Universal Robots PolyScope program: AutoGrind02.urp

Program AutoGrind02 (installation=default directory=/programs/AutoGrind createdIn=5.7.0.90932 lastSavedIn=5.11.11.1010533 robotSerialNumber=20195501059)
Calibrated DH parameters: a=[0.000146, -0.418764, -0.053981, 0.000058, -0.000023, 0]; d=[0.162545, 37.319448, -206.067439, 168.881546, 0.09955, 0.099464]; alpha=[1.57004, -0.001979, 0.002304, 1.570607, -1.57066, 0]; deltaTheta=[0, -0.174616, -1.258233, 1.432844, -0.000001, 0]
BeforeStart
  Script file /programs/AutoGrind/agscript_util-2.script
    | # File: agscript_util-2.scripts
    | # Project: AutoGrind
    | # Author: Ned Lecky, Lecky Engineering LLC
    | # Purpose: General utility function used in AutoGrind
    | 
    | global robot_util_version = "Rev 2 2022-06-02"
    | 
    | # Return max of 2 numeric values
    | def max(n1, n2):
    |   if n1 > n2:
    |     return n1
    |   else:
    |     return n2
    |   end
    | end
    | 
    | # Return min of 2 numeric values
    | def min(n1, n2):
    |   if n1 < n2:
    |     return n1
    |   else:
    |     return n2
    |   end
    | end
    | 
    | # Return absolute value of a numeric value
    | def abs(n):
    |   if n < 0:
    |     return -n
    |   else:
    |     return n
    |   end
    | end
    | 
    | # Return param limited to lowLim <= param <= hiLim
    | def limiter(param, loLim, hiLim):
    |   if param < loLim:
    |     return loLim
    |   elif param > hiLim:
    |     return hiLim
    |   else:
    |     return param
    |   end
    | end
    | 
    | # Send LF out the socket
    | def socket_send_lf():
    |   socket_send_byte(10)
    | end
    | 
    | # Send n-vectors back to socket as [n,n,n,n,n,n]
    | def return_vector(p, n = 6):
    |   socket_send_string("[")
    |   i = 0
    |   while i < n:
    |     if i > 0:
    |       socket_send_string(",")
    |     end
    |     socket_send_string(p[i])
    |     i = i + 1
    |   end
    |   socket_send_string("]")
    | end
    | 
    | # Send 6-element position back to socket as:
    | #   (isPose=False)  name=[n,n,n,n,n,n]
    | #   (isPose=True)   name=p[n,n,n,n,n,n]
    | def return_position(name, isPose, p):
    |   socket_send_string(name)
    |   socket_send_string("=")
    |   if isPose == True:
    |     socket_send_string("p")
    |   end
    |   return_vector(p, 6)
    |   socket_send_lf()
    | end
    | 
    | # Return a 6-element vector to socket as a pose name=p[.....]
    | def return_pose(name, p):
    |   return_position(name, True, p)
    | end
    | 
    | # Return a 6-element vector to socket as joint angles name=[.....]
    | def return_joints(name, p):
    |   return_position(name, False, p)
    | end
    | 
    | # Special support to receive 1-4 port,value pairs and always pad with -1s to make 4 pairs
    | # Essentialy returns command[3:end] padded out with -1s to always be 8 elements
    | # Assumes length of command is specified in command[0]
    | def command_3_padded_8(command):
    |   ret8 = [-1, -1, -1, -1, -1, -1, -1, -1]
    |   i = 0
    |   while i < command[0]-2:
    |     ret8[i] = command[i + 3]
    |     i = i + 1
    |   end
    |   return ret8
    | end
  Script file /programs/AutoGrind/agscript_robot-2.script
    | # File: agscript_robot-2.script
    | # Project: AutoGrind
    | # Author: Ned Lecky, Lecky Engineering LLC
    | # Purpose: Robot control commands supporting the AutoGrind application
    | 
    | global robot_version = "Rev 2 2022-06-07"
    | 
    | global response = "unknown"
    | global robot_index = 0
    | global robot_checkvalue = 0
    | 
    | global robot_linear_speed_mps = 0.2
    | global robot_linear_accel_mpss = 0.4
    | global robot_blend_radius_m = 0.003
    | global robot_joint_speed_rps = 1.0
    | global robot_joint_accel_rpss = 4.0
    | global robot_tcp = p[0, 0, 0.175, 0, 0, 0]
    | global robot_tcp_part = robot_tcp
    | global robot_payload_mass_kg = 1.0
    | global robot_payload_cog_m = [0, 0, 0.50]
    | # Geometry [1=FLAT 2=CYL 3=SPHERE, diameter_mm)
    | global robot_part_geometry = [0, 0]
    | global robot_door_closed_input = [-1, -1]
    | global robot_footswitch_pressed_input = [-1, -1]
    | global robot_tool_on_outputs = [-1, -1, -1, -1, -1, -1, -1, -1]
    | global robot_tool_off_outputs = [-1, -1, -1, -1, -1, -1, -1, -1]
    | global robot_coolant_on_outputs = [-1, -1, -1, -1, -1, -1, -1, -1]
    | global robot_coolant_off_outputs = [-1, -1, -1, -1, -1, -1, -1, -1]
    | global robot_freedrive_mode = 0
    | 
    | # command should be[nElements,index,checkval,param[0],param[1],...]
    | # put index into robot_index
    | # validate checkval
    | # Remove both from command so we get command = [nElements-2, param[0], param[1],...]
    | #global command = [0., 0., 0., 0., 0., 0., 0., 0., 0., 0., 0., 0., 0.]
    | def command_validate():
    |   # must be at least index, check, and 1 param
    |   if command[0] < 3:
    |     command[0] = 0
    |     return False
    |   end
    | 
    |   # Now make sure checksum matches what we expect
    |   global test_index = command[1]
    |   global test_checksum = command[2]
    |   if test_checksum != 1000 - test_index:
    |     command[0] = 0
    |     return False
    |   end
    | 
    |   # Now if we are still in the grind state and we are not getting a grind command (40) make sure we're are off the part!
    |   if grind_process_state and command[3] != 40:
    |     # Using set_grind_process_state which assumes robot_tcp_part!
    |     iset_tcp(robot_tcp_part)
    |     set_grind_process_state(False)
    |     iset_tcp(robot_tcp)
    |   end
    | 
    |   # Slide the robot commands and parameters back in command[] to remove the index and checksum
    |   local i = 3
    |   while (i < command[0] + 1):
    |     command[i-2] = command[i]
    |     i = i + 1
    |   end
    |   command[i-1] = 0
    |   command[i-2] = 0
    |   command[0] = command[0] - 2    # 2 fewer elements in the array now!
    | 
    |   global robot_index = test_index
    |   return True
    | end
    | 
    | # Call this when starting command execution
    | def command_start():
    |   global last_comand = command
    | 
    |   # This one signifies we're starting a new command!
    |   global robot_starting = robot_index
    |   socket_set_var("robot_starting", robot_starting)
    |   socket_send_line("robot_ready=False")
    | end
    | 
    | # Call this when a command is complete
    | def command_finish():
    |   local retval = "robot_response=" + response + "#robot_ready=True"
    |   socket_send_line(retval)
    | 
    |   global robot_completed = robot_index
    |   socket_set_var("robot_completed", robot_completed)
    | end
    | 
    | # Set variable interface. Interprets command[2] to select what to set and returns result to socket
    | # Can also be used for validation and enforcing limits
    | def set_variable():
    |   if command[2] == 1:
    |     # Set speed to s if s>0. Always returns current value
    |     s = command[3]
    |     if s > 0:
    |       robot_linear_speed_mps = ceil(s) / 1000.0
    |     end
    |     socket_set_var("robot_linear_speed_mmps", robot_linear_speed_mps * 1000.0)
    |     global response = "set_linear_speed()"
    |   elif command[2] == 2:
    |     # Set accel to a if a>0. Always returns current value
    |     a = command[3]
    |     if a > 0:
    |       robot_linear_accel_mpss = ceil(a) / 1000.0
    |     end
    |     socket_set_var("robot_linear_accel_mmpss", robot_linear_accel_mpss * 1000.0)
    |     global response = "set_linear_accel()"
    |   elif command[2] == 3:
    |     # Set blend to b if b>=0. Always returns current value
    |     b = command[3]
    |     if b >= 0:
    |       robot_blend_radius_m = b / 1000.0
    |     end
    |     socket_send_string("robot_blend_radius_mm=")
    |     socket_send_string(robot_blend_radius_m * 1000.0)
    |     socket_send_lf()
    |     global response = "set_blend_radius()"
    |   elif command[2] == 4:
    |     # Set joint speed to s if s>0. Always returns current value
    |     s = command[3]
    |     if s > 0:
    |       robot_joint_speed_rps = d2r(ceil(s))
    |     end
    |     socket_set_var("robot_joint_speed_dps", r2d(robot_joint_speed_rps))
    |     global response = "set_joint_speed()"
    |   elif command[2] == 5:
    |     # Set joint accel to a if a>0. Always returns current value
    |     a = command[3]
    |     if a > 0:
    |       robot_joint_accel_rpss = d2r(ceil(a))
    |     end
    |     socket_set_var("robot_joint_accel_dpss", r2d(robot_joint_accel_rpss))
    |     global response = "set_joint_accel()"
    |   elif command[2] == 6:
    |     # Set part_geometry to [shape, diameter_mm] if shape==1,2,3. Always returns "robot_part_geometry=[current geometry]"
    |     # Also updates robot_part_tcp using update_robot_tcp_part
    |     shape = command[3]
    |     if shape == 1:
    |       robot_part_geometry = [1, 0]
    |     elif shape == 2 or shape == 3:
    |       diameter_mm = limiter(command[4], 50, 3000)
    |       robot_part_geometry = [shape, diameter_mm]
    |     end
    | 
    |     update_robot_tcp_part()
    | 
    |     socket_send_string("robot_part_geometry=")
    |     return_vector(robot_part_geometry, 2)
    |     socket_send_lf()
    |     global response = "set_part_geometry()"
    |   elif command[2] == 10:
    |     # Set door closed input
    |     if command[3] >= 0:
    |       robot_door_closed_input[0] = command[3]
    |       robot_door_closed_input[1] = command[4]
    |     end
    | 
    |     socket_send_string("robot_door_closed_input=")
    |     return_vector(robot_door_closed_input, 2)
    |     socket_send_lf()
    |     socket_set_var("robot_door_closed", is_door_closed())
    |     global response = "set_door_closed_input()"
    |   elif command[2] == 11:
    |     # Set tool on output
    |     robot_tool_on_outputs = command_3_padded_8(command)
    | 
    |     socket_send_string("robot_tool_on_outputs=")
    |     return_vector(robot_tool_on_outputs, 8)
    |     socket_send_lf()
    |     global response = "set_tool_on_outputs()"
    |   elif command[2] == 12:
    |     # Set tool off output
    |     robot_tool_off_outputs = command_3_padded_8(command)
    | 
    |     socket_send_string("robot_tool_off_outputs=")
    |     return_vector(robot_tool_off_outputs, 8)
    |     socket_send_lf()
    |     global response = "set_tool_off_outputs()"
    |   elif command[2] == 13:
    |     # Set coolant on output
    |     robot_coolant_on_outputs = command_3_padded_8(command)
    | 
    |     socket_send_string("robot_coolant_on_outputs=")
    |     return_vector(robot_coolant_on_outputs, 8)
    |     socket_send_lf()
    |     global response = "set_coolant_on_outputs()"
    |   elif command[2] == 14:
    |     # Set coolant off output
    |     robot_coolant_off_outputs = command_3_padded_8(command)
    | 
    |     socket_send_string("robot_coolant_off_outputs=")
    |     return_vector(robot_coolant_off_outputs, 8)
    |     socket_send_lf()
    |     global response = "set_coolant_off_outputs()"
    |   elif command[2] == 15:
    |     # tool_on
    |     tool_power(True, 2)
    |     global response = "tool_on()"
    |   elif command[2] == 16:
    |     # tool_off
    |     tool_power(False, 2)
    |     global response = "tool_off()"
    |   elif command[2] == 17:
    |     # coolant_on
    |     coolant_flow(True, 2)
    |     global response = "coolant_on()"
    |   elif command[2] == 18:
    |     # coolant_off
    |     coolant_flow(False, 2)
    |     global response = "coolant_off()"
    |   elif command[2] == 19:
    |     # freedrive 1=on/0=off, 0=base|1=tcp|2=tcp_part, 6 axisEnables
    |     if command[3] == 0:
    |       end_freedrive_mode()
    |       iset_tcp(robot_tcp)
    |       robot_freedrive_mode = 0
    |       socket_set_var("robot_freedrive_mode", robot_freedrive_mode)
    |     else:
    |       local coordSys = command[4]
    |       local freeAxes = [command[5], command[6], command[7], command[8], command[9], command[10]]
    |       if coordSys == 1:
    |         iset_tcp(robot_tcp)
    |         freedrive_mode(freeAxes = freeAxes, feature = "tool")
    |       elif coordSys == 2:
    |         iset_tcp(robot_tcp_part)
    |         freedrive_mode(freeAxes = freeAxes, feature = "tool")
    |       else:
    |         # Base
    |         freedrive_mode(freeAxes = freeAxes)
    |       end
    |       robot_freedrive_mode = 1
    |       socket_set_var("robot_freedrive_mode", robot_freedrive_mode)
    |     end
    |     global response = "freedrive_mode()"
    |   elif command[2] == 20:
    |     # set_tcp if command[3] > -10. Always returns robot_tcp=p[...]
    |     if command[3] > -10:
    |       robot_tcp = p[command[3], command[4], command[5], command[6], command[7], command[8]]
    |       iset_tcp(robot_tcp)
    |     end
    |     return_pose("robot_tcp", get_tcp_offset())
    |     # Recompute robot_tcp_part based on current geometry
    |     update_robot_tcp_part()
    |     global response = "set_tcp()"
    |   elif command[2] == 21:
    |     # set_payload if command[3] > 0. Always return robot_m and robot_cog
    |     if command[3] > 0:
    |       robot_payload_mass_kg = command[3]
    |       robot_payload_cog_m = [command[4], command[5], command[6]]
    |       iset_payload(robot_payload_mass_kg, robot_payload_cog_m)
    |     end
    |     socket_set_var("robot_payload_mass_kg", robot_payload_mass_kg)
    |     socket_send_string("robot_payload_cog_m=")
    |     return_vector(robot_payload_cog_m, 3)
    |     socket_send_lf()
    |     global response = "set_payload()"
    |   elif command[2] == 22:
    |     # Set footswitch pressed input
    |     if command[3] >= 0:
    |       robot_footswitch_pressed_input[0] = command[3]
    |       robot_footswitch_pressed_input[1] = command[4]
    |     end
    | 
    |     socket_send_string("robot_footswitch_pressed_input=")
    |     return_vector(robot_footswitch_pressed_input, 2)
    |     socket_send_lf()
    |     socket_set_var("robot_footswitch_pressed", is_footswitch_pressed())
    |     global response = "set footswitch_pressed_input()"
    |   elif command[2] == 30:
    |     # set_output
    |     local out = command[3]
    |     local state = command[4] > 0
    |     set_digital_out(out, state)
    |     global response = "set_output()"
    |   else:
    |     global response = "set_variable ERROR"
    |   end
    | end
    | 
    | # Compute appropriate robot_tcp for the part based on robot_tcp and robot_part_geometry
    | # They're the same for flat parts, but the TCP is adjusted to the center of the cylinder or sphere
    | def update_robot_tcp_part():
    |   shape = robot_part_geometry[0]
    |   if shape == 1:  # Flat
    |     robot_tcp_part = robot_tcp
    |   else:  # Cylinder or Sphere
    |     robot_tcp_part = pose_trans(robot_tcp, p[0, 0, robot_part_geometry[1] / 2000.0, 0, 0, 0])
    |   end
    |   return_pose("robot_tcp_part", robot_tcp_part)
    | end
    | 
    | # Send get_tcp_offset() result to socket
    | def return_tcp_offset():
    |   p = get_tcp_offset()
    |   return_pose("tcp_offset", p)
    |   global response = "return_tcp_offset()"
    | end
    | 
    | # Send get_actual_tcp_pose() to socket
    | def return_actual_tcp_pose():
    |   p = iget_actual_tcp_pose()
    |   return_pose("actual_tcp_pose", p)
    |   global response = "return_actual_tcp_pose()"
    | end
    | 
    | # Send get_actual_joint_positions() to socket
    | def return_get_actual_joint_positions():
    |   p = iget_actual_joint_positions()
    |   return_joints("actual_joint_positions", p)
    |   global response = "return_get_actual_joint_positions()"
    | end
    | 
    | # Send both joints and pose to socket labeled position_p and position_q
    | def return_both_positions():
    |   return_joints("position_q", iget_actual_joint_positions())
    |   return_pose("position_p", iget_actual_tcp_pose())
    |   global response = "return_both_positions()"
    | end
    | 
    | # Movel relatively in base coordinates
    | def movel_relative_base(p1):
    |   local p0 = get_target_tcp_pose()
    |   local p2 = pose_add(p0, p1)
    |   if p1[0] == 0 and p1[1] == 0 and p1[2] == 0:  # Rotational move
    |     imovel(p2, robot_joint_accel_rpss, robot_joint_speed_rps)
    |   else:
    |     imovel(p2, robot_linear_accel_mpss, robot_linear_speed_mps)
    |   end
    |   global response = "movel_relative_base()"
    | end
    | 
    | # Movel relatively in TCP coordinates
    | def movel_relative_tcp(p1):
    |   local p2 = pose_trans(get_target_tcp_pose(), p1)
    |   if p1[0] == 0 and p1[1] == 0 and p1[2] == 0:  # Rotational move
    |     imovel(p2, robot_joint_accel_rpss, robot_joint_speed_rps)
    |   else:
    |     imovel(p2, robot_linear_accel_mpss, robot_linear_speed_mps)
    |   end
    |   global response = "movel_relative_tcp()"
    | end
    | 
    | # Movel relatively in TCP_part coordinates
    | def movel_relative_tcp_part(p1):
    |   iset_tcp(robot_tcp_part)
    |   local p2 = pose_trans(get_target_tcp_pose(), p1)
    |   if p1[0] == 0 and p1[1] == 0 and p1[2] == 0:  # Rotational move
    |     imovel(p2, robot_joint_accel_rpss, robot_joint_speed_rps)
    |   else:
    |     imovel(p2, robot_linear_accel_mpss, robot_linear_speed_mps)
    |   end
    |   iset_tcp(robot_tcp)
    |   global response = "movel_relative_tcp_part()"
    | end
    | 
    | # Change one element of current pose and movel there
    | def movel_one_only(index = 0, val = 0):
    |   local p = get_target_tcp_pose()
    |   p[index] = val
    |   if index < 3:  # Translational
    |     imovel(p, a = robot_linear_accel_mpss, v = robot_linear_speed_mps)
    |   else:
    |     imovel(p, a = robot_joint_accel_rpss, v = robot_joint_speed_rps)
    |   end
    |   global response = "movel_one_only()"
    | end
    | 
    | # Change only rotation elements of current pose and movel there
    | def movel_rot_only(r1 = 0, r2 = 0, r3 = 0):
    |   local p = get_target_tcp_pose()
    |   p[3] = r1
    |   p[4] = r2
    |   p[5] = r3
    |   imovel(p, a = robot_joint_accel_rpss, v = robot_joint_speed_rps)
    |   global response = "movel_rot_only()"
    | end
    | 
    | # Movej to position (works with joints or poses)
    | def movej_ag(p):
    |   imovej(p, a = robot_joint_accel_rpss, v = robot_joint_speed_rps)
    |   global response = "movej_ag()"
    | end
    | 
    | # Movel to position (works with joints or poses)
    | def movel_ag(p):
    |   imovel(p, a = robot_linear_accel_mpss, v = robot_linear_speed_mps)
    |   global response = "movel_ag()"
    | end
    | 
    | # ####################################################################################
    | # Interrupting Motion
    | # Motion and force_mode and part contact muct all end if any of 3 things happen
    | #  1) Door is opened
    | #  2) We're in contact with the part and grinding, but no grind command comes within some time (default 1.5s)
    | #  3) We receive an abort message from the host
    | #
    | # How is it implemented?
    | #
    | # 1) io_monitor_thread (below) is ALWAYS running. Fires every time_door_check_rate_s (0.25s)
    | #    - Whenever it sees the state of the door change, it sends SET robot_door_closed state to host
    | #    - Whenever it sees the state of the footswitch (DIN7) change, it sends SET robot_footswitch state to host
    | #    - It monitors if we're still in contact wth the part butr not grinding (grind_process_state and grind_ready)
    | #      - If that goes beyond grind_max_wait_ms it sets halt_grind=True
    | # 2) no_command function (below). Called by PolScript everyu time it's waiting for a command and doesn't get one with a second
    | #    - If halt_grind is set (by door monitor thread above)
    | #      - stopl and simulate receiving a grind_retract
    | #      - THIS FORCES THE force_off and motion commands to come from the primary thread, as they must
    | # 3) listener_thread started by grind()
    | #    - This runs only while a grind is in progress
    | #    - It listens for commands from the host since PolyScope is blocked
    | #    - Any command received increments halt_count which makes ok_to_proceed() false
    | #    - That is checked in all the grinding programs and forces them to finish up and get off the part in an orderly fashion
    | 
    | # ####################################################################################
    | # START AUTOMATED DOOR MONITORING THREAD
    | #
    | # Return True if door in closed state (or if door input is undefined)
    | def is_door_closed():
    |   if robot_door_closed_input[0] < 0:
    |     return True
    |   end
    |   if get_standard_digital_in(robot_door_closed_input[0]):
    |     f = 1
    |   else:
    |     f = 0
    |   end
    |   return f == robot_door_closed_input[1]
    | end
    | 
    | # Return True if footswitch pressed (or False if footswitch input is undefined)
    | def is_footswitch_pressed():
    |   if robot_footswitch_pressed_input[0] < 0:
    |     return False
    |   end
    |   if get_standard_digital_in(robot_footswitch_pressed_input[0]):
    |     f = 1
    |   else:
    |     f = 0
    |   end
    |   return f == robot_footswitch_pressed_input[1]
    | end
    | 
    | global robot_door_closed = is_door_closed()
    | global robot_footswitch_pressed = is_footswitch_pressed()
    | global time_in_uncommanded_grind = 0
    | global time_door_check_rate_s = 0.250
    | global grind_max_wait_ms = 1500
    | # Also monitors footswitch!
    | thread io_monitor_thread():
    |   # Send current state on start... in future will only be sent on change
    |   socket_set_var("robot_door_closed", robot_door_closed)
    |   socket_set_var("robot_footswitch_pressed", robot_footswitch_pressed)
    | 
    |   while True:
    |     sleep(time_door_check_rate_s)
    |     local new_door_closed = is_door_closed()
    |     local new_footswitch_pressed = is_footswitch_pressed()
    | 
    |     # Notify host if door state has changed
    |     if robot_door_closed != new_door_closed:
    |       robot_door_closed = new_door_closed
    |       socket_set_var("robot_door_closed", robot_door_closed)
    |     end
    | 
    |     # Notify host if footswitch state has changed
    |     if robot_footswitch_pressed != new_footswitch_pressed:
    |       robot_footswitch_pressed = new_footswitch_pressed
    |       socket_set_var("robot_footswitch_pressed", robot_footswitch_pressed)
    |     end
    | 
    |     # Check for still in grind process but not executing a grind command
    |     # This is what happens after a grind_...(....,1) executes while waiting for next command
    |     if grind_process_state and grind_ready:
    |       time_in_uncommanded_grind = time_in_uncommanded_grind + time_door_check_rate_s
    |       # No new grind commands for grind_max_wait_ms... schedule a grind_retract!
    |       if time_in_uncommanded_grind > grind_max_wait_ms / 1000.0:
    |         global halt_grind = True
    |       end
    |     else:
    |       time_in_uncommanded_grind = 0
    |     end
    |   end
    | end
    | global ioMonitorThread = run io_monitor_thread()
    | #
    | # END AUTOMATED DOOR MONITORING THREAD
    | # ####################################################################################
    | 
    | # ####################################################################################
    | # START NO_COMMAND HOUSEKEEPING
    | # This gets called when the PolyScope receives no command (about 1/second)
    | # We can fire off any command here safely since no others will be seen until we exit
    | #
    | global no_command_count = 0
    | global halt_grind = False
    | def no_command():
    |   global no_command_count = no_command_count + 1
    | 
    |   if grind_process_state and grind_ready and halt_grind:
    |     halt_grind = False
    |     istopl(20)
    | 
    |     iset_tcp(robot_tcp_part)
    |     set_grind_process_state(False)
    |     iset_tcp(robot_tcp)
    |   end
    | end
    | #
    | # END NO_COMMAND HOUSEKEEPING
    | # ####################################################################################
    | 
    | # ####################################################################################
    | # START TOUCHOFF HANDLER
    | #
    | def calculate_point_to_move_towards(feature, direction, position_distance):
    |   local posDir = [direction[0], direction[1], direction[2]]
    |   if (norm(posDir) < 1e-6):
    |     return get_target_waypoint()
    |   end
    |   local direction_vector_normalized = normalize(posDir)
    |   local displacement_pose = p[direction_vector_normalized[0] * position_distance, direction_vector_normalized[1] * position_distance, direction_vector_normalized[2] * position_distance, 0, 0, 0]
    |   local wanted_displacement_in_base_frame = pose_sub(pose_trans(feature, displacement_pose), feature)
    |   return pose_add(get_target_waypoint(), wanted_displacement_in_base_frame)
    | end
    | #$ 7 "Robot Program"
    | #$ 8 "MoveL"
    | #$ 9 "Direction: Tool Z+"
    | global move_thread_flag = 0
    | global move_thread_approach_speed_mps = 0.01
    | thread move_thread():
    |   enter_critical
    |   move_thread_flag = 1
    |   local towardsPos = calculate_point_to_move_towards(get_forward_kin(), [0.0, 0.0, 1.0], 0.025)
    |   imovel(towardsPos, a = 0.5, v = move_thread_approach_speed_mps)
    |   move_thread_flag = 2
    |   exit_critical
    | end
    | 
    | # Currently using speed_mmps for both approach and 2X for departure
    | def touchoff(approach_speed_mmps, retract_mm):
    |   approach_speed_mps = approach_speed_mmps / 1000.0
    |   global move_thread_approach_speed_mps = approach_speed_mps
    | 
    |   retract_speed_mps = approach_speed_mps * 2.0
    | 
    |   retract_m = retract_mm / 1000.0
    | 
    |   move_thread_flag = 0
    |   move_thread_han = run move_thread()
    |   while (True):
    |     local targetTcpDirection = get_target_tcp_speed()
    |     local stepsToRetract = tool_contact(direction = targetTcpDirection)
    |     if (stepsToRetract > 0):
    |       kill move_thread_han
    |       imover_restart()
    |       istopl(20)
    |       local backTrackMovement = get_actual_joint_positions_history(stepsToRetract)
    |       local contactPose = get_forward_kin(backTrackMovement)
    |       local posDir = [targetTcpDirection[0], targetTcpDirection[1], targetTcpDirection[2]]
    |       local retractTo = contactPose
    |       if (norm(posDir) > 1e-6):
    |         local normalizedPosDir = normalize(posDir)
    |         local additionalRetraction = p[normalizedPosDir[0] * retract_m, normalizedPosDir[1] * retract_m, normalizedPosDir[2] * retract_m, 0, 0, 0]
    |         retractTo = pose_sub(contactPose, additionalRetraction)
    |       end
    |       imovel(retractTo, a = 1.0, v = retract_speed_mps)
    |       #$ 10 "Until (tool_contact_detection)"
    |       return True
    |       break
    |     end
    |     sleep(1.0E-10)
    |     if (move_thread_flag > 1):
    |       join move_thread_han
    |       #$ 11 "Until (distance)"
    |       #$ 12 "Popup: No part encountered"
    |       #popup("No part encountered", "Message", False, False, blocking = True)
    |       return False
    |       break
    |     end
    |     sync()
    |   end
    |   return False
    | end
    | #
    | # END TOUCHOFF HANDLER
    | # ####################################################################################
    | 
    | # ####################################################################################
    | # START IMOVER SYSTEM
    | #
    | global imover_realtime_enabled = True
    | global imover_p = p[0, 0, 0, 0, 0, 0]
    | global imover_q = [0, 0, 0, 0, 0, 0]
    | global imover_a = 1.2
    | global imover_v = 0.25
    | global imover_t = 0
    | global imover_r = 0
    | global imover_f = False
    | global imover_tcp = p[0, 0, 0, 0, 0, 0]
    | global imover_mass = 1.0
    | global imover_cog = [0, 0, 0]
    | global imover_thread_handle = 0
    | global imover_cmd = 0
    | global imover_cmd_hist = [0, 0, 0, 0, 0, 0, 0, 0, 0, 0]
    | global imover_param1 = 0
    | global imover_param2 = 0
    | imover_PING = 1
    | imover_MOVEL = 2
    | imover_MOVEJ = 3
    | imover_STOPL = 4
    | imover_STARTFORCE = 5
    | imover_UPDATEFORCE = 6
    | imover_ENDFORCE = 7
    | imover_GETACTUALTCPPOSE = 8
    | imover_GETACTUALJOINTPOSITIONS = 9
    | imover_SETTCP = 10
    | imover_SETPAYLOAD = 11
    | imover_TOUCHOFF = 12
    | 
    | def imover_realtime(f = False):
    |   if f and not imover_realtime_enabled:
    |     imover_realtime_enabled = True
    |     imover_restart()
    |   elif not f and imover_realtime_enabled:
    |     imover_abort()
    |     imover_realtime_enabled = False
    |   end
    | end
    | 
    | def imover_abort():
    |   if not imover_realtime_enabled:
    |     return None
    |   end
    | 
    |   if imover_thread_handle > 0:
    |     kill imover_thread_handle
    |     imover_thread_handle = 0
    |   end
    |   set_tcp(imover_tcp)
    |   set_payload(imover_mass, imover_cog)
    | end
    | 
    | def imover_restart():
    |   if not imover_realtime_enabled:
    |     return None
    |   end
    | 
    |   imover_abort()
    |   global imover_thread_handle = run imover_thread()
    |   iset_tcp(imover_tcp)
    |   iset_payload(imover_mass, imover_cog)
    | end
    | 
    | def imover_wait(terminate_not_ok = False):
    |   while imover_cmd > 0:
    |     if terminate_not_ok and not ok_to_proceed():
    |       return None
    |     end
    |     sync()
    |   end
    | end
    | 
    | def imover_cmd_exec(cmd, param1 = 0, param2 = 0, terminate_not_ok = False, no_wait = False):
    |   imover_wait()
    |   global imover_param1 = param1
    |   global imover_param2 = param2
    | 
    |   local i = 9
    |   while i > 0:
    |     imover_cmd_hist[i] = imover_cmd_hist[i - 1]
    |     i = i - 1
    |   end
    |   imover_cmd_hist[0] = cmd
    |   global imover_cmd = cmd
    | 
    |   if not no_wait:
    |     imover_wait(terminate_not_ok)
    |   end
    | end
    | 
    | def istopl(a, aRot = 999):
    |   if imover_realtime_enabled:
    |     imover_cmd_exec(imover_STOPL, a, aRot)
    |   else:
    |     if aRot == 999:
    |       stopl(a)
    |     else:
    |       stopl(a, aRot)
    |     end
    |   end
    | end
    | 
    | def iforce_mode(force_n, approach_speed_mmps):
    |   if imover_realtime_enabled:
    |     imover_cmd_exec(imover_STARTFORCE, force_n, approach_speed_mmps)
    |   else:
    |     sleep(0.25)
    |     zero_ftsensor()
    | 
    |     # Using the defaults here
    |     force_mode_set_damping(0)
    |     force_mode_set_gain_scaling(1)
    | 
    |     # Force is in tool frame
    |     # Compliant in Tool Z
    |     # Applying grind_force_n in Z+
    |     # 2: Force frame not transformed
    |     # Speed limits
    |     force_mode(tool_pose(), [0, 0, 1, 0, 0, 0], [0.0, 0.0, force_n, 0.0, 0.0, 0.0], 2, [0.1, 0.1, approach_speed_mmps / 1000.0, 0.3490658503988659, 0.3490658503988659, 0.3490658503988659])
    |   end
    | end
    | 
    | def iforce_update(force_n = 5, approach_speed_mmps = 10):
    |   if imover_realtime_enabled:
    |     imover_cmd_exec(imover_UPDATEFORCE, force_n, approach_speed_mmps)
    |   else:
    |     # Force is in tool frame
    |     # Compliant in Tool Z
    |     # Applying grind_force_n in Z+
    |     # 2: Force frame not transformed
    |     # Speed limits
    |     force_mode(tool_pose(), [0, 0, 1, 0, 0, 0], [0.0, 0.0, force_n, 0.0, 0.0, 0.0], 2, [0.1, 0.1, approach_speed_mmps / 1000.0, 0.3490658503988659, 0.3490658503988659, 0.3490658503988659])
    |   end
    | end
    | 
    | def iend_force_mode():
    |   if imover_realtime_enabled:
    |     imover_cmd_exec(imover_ENDFORCE)
    |   else:
    |     end_force_mode()
    |   end
    | end
    | 
    | def iget_actual_tcp_pose():
    |   if imover_realtime_enabled:
    |     imover_cmd_exec(imover_GETACTUALTCPPOSE)
    |     return imover_p
    |   else:
    |     return get_actual_tcp_pose()
    |   end
    | end
    | 
    | def iget_actual_joint_positions():
    |   if imover_realtime_enabled:
    |     imover_cmd_exec(imover_GETACTUALJOINTPOSITIONS)
    |     return imover_q
    |   else:
    |     return get_actual_joint_positions()
    |   end
    | end
    | 
    | def iset_tcp(tcp):
    |   imover_tcp = tcp
    |   if imover_realtime_enabled:
    |     imover_cmd_exec(imover_SETTCP)
    |   else:
    |     set_tcp(tcp)
    |   end
    | end
    | 
    | def iset_payload(mass, cog):
    |   imover_mass = mass
    |   imover_cog = cog
    |   if imover_realtime_enabled:
    |     imover_cmd_exec(imover_SETPAYLOAD)
    |   else:
    |     set_payload(mass, cog)
    |   end
    | end
    | 
    | def itouchoff(speed_mmps, retract_mm):
    |   if False: #imover_realtime_enabled:
    |     imover_param1 = speed_mmps
    |     imover_param2 = retract_mm
    |     imover_cmd_exec(imover_TOUCHOFF)
    |     return imover_f
    |   else:
    |     return touchoff(speed_mmps, retract_mm)
    |   end
    | end
    | 
    | def imovel(p, a = 1.2, v = 0.25, t = 0, r = 0):
    |   if imover_realtime_enabled:
    |     imover_wait()
    |     global imover_p = p
    |     global imover_a = a
    |     global imover_v = v
    |     global imover_t = t
    |     global imover_r = r
    |     imover_cmd_exec(imover_MOVEL, 0, 0, True)
    |   else:
    |     movel(p, a = a, v = v, t = t, r = r)
    |   end
    | end
    | 
    | def imovel_int(p, a = 1.2, v = 0.25, t = 0, r = 0, no_wait = False):
    |   if not ok_to_proceed():
    |     return None
    |   end
    | 
    |   if imover_realtime_enabled:
    |     imover_wait()
    |     global imover_p = p
    |     global imover_a = a
    |     global imover_v = v
    |     global imover_t = t
    |     global imover_r = r
    |     imover_cmd_exec(imover_MOVEL, 0, 0, True, no_wait)
    |     if not ok_to_proceed():
    |       imover_restart()
    |       istopl(grind_accel_mpss, grind_rot_accel_rpss)
    |     end
    |   else:
    |     movel(p, a = a, v = v, t = t, r = r)
    |   end
    | end
    | 
    | def imovej(q, a = 1.2, v = 0.25, t = 0, r = 0):
    |   if imover_realtime_enabled:
    |     imover_wait()
    |     global imover_q = q
    |     global imover_a = a
    |     global imover_v = v
    |     global imover_t = t
    |     global imover_r = r
    |     imover_cmd_exec(imover_MOVEJ, 0, 0, True)
    |   else:
    |     movej(q, a = a, v = v, t = t, r = r)
    |   end
    | end
    | 
    | thread imover_thread():
    |   global imover_cmd = 0
    |   while True:
    |     if imover_cmd == imover_MOVEL:
    |       movel(imover_p, a = imover_a, v = imover_v, t = imover_t, r = imover_r)
    |       global imover_cmd = 0
    |     elif imover_cmd == imover_MOVEJ:
    |       movej(imover_q, imover_a, imover_v, imover_t, imover_r)
    |       global imover_cmd = 0
    |     elif imover_cmd == imover_STOPL:
    |       stopl(grind_speed_mps, grind_rot_speed_rps)
    |       global imover_cmd = 0
    |     elif imover_cmd == imover_STARTFORCE:
    |       # Settle and zero the force/torque sensor
    |       sleep(0.25)
    |       zero_ftsensor()
    | 
    |       # Using the defaults here
    |       force_mode_set_damping(0)
    |       force_mode_set_gain_scaling(1)
    | 
    |       # Force is in tool frame
    |       # Compliant in Tool Z
    |       # Applying grind_force_n in Z+
    |       # 2: Force frame not transformed
    |       # Speed limits
    |       force_mode(tool_pose(), [0, 0, 1, 0, 0, 0], [0.0, 0.0, imover_param1, 0.0, 0.0, 0.0], 2, [0.1, 0.1, imover_param2 / 1000.0, 0.3490658503988659, 0.3490658503988659, 0.3490658503988659])
    |       global imover_cmd = 0
    |     elif imover_cmd == imover_UPDATEFORCE:
    |       # Update force
    |       # Force is in tool frame
    |       # Compliant in Tool Z
    |       # Applying grind_force_n in Z+
    |       # 2: Force frame not transformed
    |       # Speed limits
    |       force_mode(tool_pose(), [0, 0, 1, 0, 0, 0], [0.0, 0.0, imover_param1, 0.0, 0.0, 0.0], 2, [0.1, 0.1, imover_param2 / 1000.0, 0.3490658503988659, 0.3490658503988659, 0.3490658503988659])
    |       global imover_cmd = 0
    |     elif imover_cmd == imover_ENDFORCE:
    |       end_force_mode()
    |       global imover_cmd = 0
    |     elif imover_cmd == imover_GETACTUALTCPPOSE:
    |       imover_p = get_actual_tcp_pose()
    |       global imover_cmd = 0
    |     elif imover_cmd == imover_GETACTUALJOINTPOSITIONS:
    |       imover_q = get_actual_joint_positions()
    |       global imover_cmd = 0
    |     elif imover_cmd == imover_SETTCP:
    |       set_tcp(imover_tcp)
    |       global imover_cmd = 0
    |     elif imover_cmd == imover_SETPAYLOAD:
    |       set_payload(imover_mass, imover_cog)
    |       global imover_cmd = 0
    |     elif imover_cmd == imover_TOUCHOFF:
    |       imover_f = touchoff(imover_param1, imover_param2)
    |       global imover_cmd = 0
    |     elif imover_cmd == imover_PING:
    |       global imover_cmd = 0
    |     end
    |     sync()
    |   end
    | end
    | global imover_thread_handle = run imover_thread()
    | #
    | # END IMOVER SYSTEM
    | # ####################################################################################
  Script file /programs/AutoGrind/agscript_grind-2.script
    | # File: agscript_grind-2.script
    | # Project: AutoGrind Code Rev 2 IMOVER
    | # Author: Ned Lecky, Lecky Engineering LLC
    | # Purpose: All grinding functions used in AutoGrind
    | 
    | global grind_version = "Rev 2 2022-06-07"
    | 
    | global grind_abort_listener_thread_handle = 0
    | global pattern_grind_thread_handle = 0
    | 
    | global halt_count = 0
    | global halt_command = [0, 0, 0, 0]
    | 
    | global grind_ready = True
    | # grind_contact_enable:  0=No Contact   1=Touch but no tool/coolant on or force  2=Touch, Tool, Coolant, and Force
    | global grind_contact_enable = 0
    | global grind_touch_retract_mm = 3       # How far to retract after touch  (we do 2X this for ghrind_contact_enable=1)
    | global grind_touch_speed_mmps = 0.1     # How fast to go in for the touch
    | global grind_force_dwell_ms = 500       # How long to dwell after turning force more on
    | global grind_max_blend_radius_m = 0.010 # Max blend radius to use while grinding
    | global grind_blend_radius_m = 0.001     # Current blend radius to use while grinding
    | global grind_trial_speed_mmps = 20      # Grinding speed when not really grinding!
    | global grind_accel_mmpss = 100          # Acceleration to use in grinding moves
    | global grind_point_frequency_hz = 4     # Points per second to generate in grind_movel
    | 
    | # Planning points
    | global p_operator_init = p[0, 0, 0, 0, 0, 0]    # Where we were when operator issued first grind command
    | global p_contact_init = p[0, 0, 0, 0, 0, 0]     # Where we first contacted the part
    | global dp_from_contact_center = p[0, 0, 0, 0, 0, 0]   # How did we offset from p_operator_int prior to contact?
    | global p_contact_center = p[0, 0, 0, 0, 0, 0]   # Computed where center of pattern would be in contact with part
    | 
    | MATH_PI = 3.1415926535
    | 
    | # Set global grind_n_cycles based on whether we really going to grind
    | def n_cycle_setter(n_cycles):
    |   if grind_contact_enable == 2:
    |     global grind_n_cycles = limiter(n_cycles, 0, 100)
    |   else:
    |     global grind_n_cycles = limiter(n_cycles, 0, 1)
    |   end
    |   socket_set_var("grind_n_cycles", grind_n_cycles)
    | end
    | 
    | # Set all speed and acceleration globals based on part geometry and whether we really going to grind
    | def speed_setter(speed_mmps, min_feature_mm, is_circle = False):
    |   speed_mmps = limiter(speed_mmps, 0.1, 200)
    | 
    |   # Figure out best blend radius to use
    |   global grind_min_feature_m = min_feature_mm / 1000.0
    |   global grind_blend_radius_m = min(grind_max_blend_radius_m, grind_min_feature_m / 4)
    |   if is_circle:
    |     if grind_blend_radius_m < 0.0015:
    |       grind_blend_radius_m = 0
    |     end
    |   else:
    |     if grind_blend_radius_m < 0.0015:
    |       grind_blend_radius_m = 0
    |     end
    |   end
    | 
    |   if grind_contact_enable == 2:
    |     global grind_speed_mps = speed_mmps / 1000.0
    |   else:
    |     global grind_speed_mps = grind_trial_speed_mmps / 1000.0
    |   end
    |   global grind_accel_mpss = grind_accel_mmpss / 1000.0
    | 
    |   # Default rotational speeds same as linear
    |   global grind_rot_speed_rps = 0
    |   global grind_rot_accel_rpss = 0
    |   global grind_rot_blend_radius_rad = 0
    | 
    |   # If part is cylinder or spherical, diameter will be >0
    |   local diam_m = robot_part_geometry[1] / 1000.0
    |   if diam_m > 0.0:
    |     # These are 1/4 the theoretical rotational speeds but we need to set them like this to get the correct speed- why??????
    |     local coeff = 0.5 # Used to be 0.5 and inexplicable
    |     global grind_rot_speed_rps = grind_speed_mps * coeff / diam_m
    |     global grind_rot_accel_rpss = grind_accel_mpss * coeff / diam_m
    |     global grind_rot_blend_radius_rad = grind_blend_radius_m * coeff / diam_m
    |   end
    | end
    | 
    | # Set grind variables chosen by command[2]
    | # Value after set is always returned to socket
    | def set_grind_variable():
    |   global grind_ready = False
    |   socket_send_line("grind_ready=False")
    | 
    |   if command[2] == 1:
    |     global response = "set grind_contact_enable"
    |     if command[3] >= 0 and command[3] <= 2:
    |       global grind_contact_enable = ceil(command[3])
    |     end
    |     socket_set_var("grind_contact_enable", grind_contact_enable)
    |   elif command[2] == 2:
    |     global response = "set grind_touch_retract_mm"
    |     if command[3] >= 0:
    |       global grind_touch_retract_mm = ceil(command[3])
    |     end
    |     socket_set_var("grind_touch_retract_mm", grind_touch_retract_mm)
    |   elif command[2] == 3:
    |     global response = "set grind_touch_speed_mmps"
    |     if command[3] >= 0:
    |       global grind_touch_speed_mmps = ceil(command[3])
    |     end
    |     socket_set_var("grind_touch_speed_mmps", grind_touch_speed_mmps)
    |   elif command[2] == 4:
    |     global response = "set grind_force_dwell_ms"
    |     if command[3] >= 0:
    |       global grind_force_dwell_ms = ceil(command[3])
    |     end
    |     socket_set_var("grind_force_dwell_ms", grind_force_dwell_ms)
    |   elif command[2] == 5:
    |     global response = "set grind_max_wait_ms"
    |     if command[3] >= 0:
    |       global grind_max_wait_ms = ceil(command[3])
    |     end
    |     socket_set_var("grind_max_wait_ms", grind_max_wait_ms)
    |   elif command[2] == 6:
    |     global response = "set grind_max_blend_radius_mm"
    |     if command[3] >= 0:
    |       global grind_max_blend_radius_m = command[3] / 1000.0
    |     end
    |     socket_send_string("grind_max_blend_radius_mm=")
    |     socket_send_string(grind_max_blend_radius_m * 1000.0)
    |     socket_send_lf()
    |   elif command[2] == 7:
    |     global response = "set grind_trial_speed_mmps"
    |     if command[3] > 0:
    |       global grind_trial_speed_mmps = ceil(command[3])
    |     end
    |     socket_set_var("grind_trial_speed_mmps", grind_trial_speed_mmps)
    |   elif command[2] == 8:
    |     global response = "set grind_accel_mmpss"
    |     if command[3] > 0:
    |       global grind_accel_mmpss = ceil(command[3])
    |     end
    |     socket_set_var("grind_accel_mmpss", grind_accel_mmpss)
    |   elif command[2] == 9:
    |     global response = "set grind_point_frequency_hz"
    |     if command[3] >= 0:
    |       global grind_point_frequency_hz = ceil(command[3])
    |     end
    |     socket_set_var("grind_point_frequency_hz", grind_point_frequency_hz)
    |   else:
    |     global response = "Unknown grind set variable command"
    |   end
    | 
    |   global grind_ready = True
    |   socket_send_line("grind_ready=True")
    | end
    | 
    | # Execute the desired grind operation as specified in command[2]...
    | def grind():
    |   global grind_ready = False
    |   socket_send_line("grind_ready=False")
    | 
    |   # Start listening for abort commands from host
    |   if grind_abort_listener_thread_handle > 0:
    |     kill grind_abort_listener_thread_handle
    |     grind_abort_listener_thread_handle = 0
    |   end
    |   grind_abort_listener_thread_handle = run grind_abort_listener_thread()
    | 
    |   global grind_cycle = 0
    |   socket_set_var("grind_cycle", grind_cycle)
    | 
    |   # Install tcp that puts tcp at center of part (noop for flat parts!)
    |   iset_tcp(robot_tcp_part)
    | 
    |   if command[2] == 10:
    |     # LINEAR GRIND
    |     global response = "grind_line"
    |     global grind_dx_mm = limiter(command[3], -1000, 1000)
    |     global grind_dy_mm = limiter(command[4], -1000, 1000)
    |     n_cycle_setter(command[5])
    |     speed_setter(command[6], 0)
    |     global grind_force_n = limiter(command[7], 0, 100)
    |     global grind_continue = command[8] > 0
    |     imover_realtime(True)
    |     grind_line(grind_dx_mm, grind_dy_mm, grind_n_cycles, grind_continue)
    | 
    |   elif command[2] == 20:
    |     # RECTANGULAR GRIND
    |     global response = "grind_rect"
    |     global grind_dx_mm = limiter(command[3], 0, 1000)
    |     global grind_dy_mm = limiter(command[4], 0, 1000)
    |     n_cycle_setter(command[5])
    |     speed_setter(command[6], min(grind_dx_mm, grind_dy_mm))
    |     global grind_force_n = limiter(command[7], 0, 100)
    |     global grind_continue = command[8] > 0
    |     imover_realtime(True)
    |     grind_rect(grind_dx_mm, grind_dy_mm, grind_n_cycles, grind_continue)
    | 
    |   elif command[2] == 30:
    |     # SERPENTINE GRIND
    |     global response = "grind_serpentine"
    |     global grind_dx_mm = limiter(command[3], 0, 1000)
    |     global grind_dy_mm = limiter(command[4], 0, 1000)
    |     global grind_n_xsteps = limiter(command[5], 1, grind_dx_mm)
    |     global grind_n_ysteps = limiter(command[6], 1, grind_dy_mm)
    |     n_cycle_setter(command[7])
    |     local min_feature_mm = min(grind_dx_mm / grind_n_xsteps, grind_dy_mm / grind_n_ysteps)
    |     speed_setter(command[8], min_feature_mm)
    |     global grind_force_n = limiter(command[9], 0, 10)
    |     global grind_continue = command[10] > 0
    |     imover_realtime(True)
    |     grind_serpentine(grind_dx_mm, grind_dy_mm, grind_n_xsteps, grind_n_ysteps, grind_n_cycles, grind_continue)
    | 
    |   elif command[2] == 40:
    |     # POLYGON GRIND
    |     global response = "grind_poly"
    |     global grind_circle1_diam_mm = limiter(command[3], 0, 1000)
    |     global grind_n_sides = limiter(command[4], 1, 1000)
    |     n_cycle_setter(command[5])
    |     local min_feature_mm = max(2, grind_circle1_diam_mm)
    |     speed_setter(command[6], min_feature_mm)
    |     global grind_force_n = limiter(command[7], 0, 100)
    |     global grind_continue = command[8] > 0
    |     imover_realtime(True)
    |     grind_poly(grind_circle1_diam_mm, grind_n_sides, grind_n_cycles, grind_continue)
    | 
    |   elif command[2] == 45:
    |     # CIRCULAR GRIND
    |     global response = "grind_circle"
    |     global grind_circle1_diam_mm = limiter(command[3], 0, 1000)
    |     n_cycle_setter(command[4])
    |     local min_feature_mm = max(2, grind_circle1_diam_mm)
    |     speed_setter(command[5], min_feature_mm, is_circle = True)
    |     global grind_force_n = limiter(command[6], 0, 100)
    |     global grind_continue = command[7] > 0
    |     imover_realtime(False)
    |     grind_circle(grind_circle1_diam_mm, grind_n_cycles, grind_continue)
    |     imover_realtime(True)
    | 
    |   elif command[2] == 50:
    |     # SPIRAL GRIND
    |     global response = "grind_spiral"
    |     global grind_circle1_diam_mm = limiter(command[3], 0, 1000)
    |     global grind_circle2_diam_mm = limiter(command[4], 0, 1000)
    |     global grind_n_revolutions = limiter(command[5], 1, 100)
    |     n_cycle_setter(command[6])
    |     local min_diam_mm = min(grind_circle1_diam_mm, grind_circle2_diam_mm)
    |     local min_feature_mm = max(2, min_diam_mm)
    |     speed_setter(command[7], min_feature_mm, is_circle = True)
    |     global grind_force_n = limiter(command[8], 0, 100)
    |     global grind_continue = command[9] > 0
    |     imover_realtime(False)
    |     grind_spiral(grind_circle1_diam_mm, grind_circle2_diam_mm, grind_n_revolutions, grind_n_cycles, grind_continue)
    |     imover_realtime(True)
    | 
    |   elif command[2] == 99:
    |     # RETRACT COMMAND
    |     global response = "grind_retract"
    |     set_grind_process_state(False)
    | 
    |   else:
    |     # Illegal grind command
    |     global response = "Unknown grind command"
    |   end
    | 
    |   # Restore tool-only tcp
    |   iset_tcp(robot_tcp)
    | 
    |   # Stop listening for abort commands from host
    |   if grind_abort_listener_thread_handle > 0:
    |     kill grind_abort_listener_thread_handle
    |     grind_abort_listener_thread_handle = 0
    |   end
    | 
    |   global grind_ready = True
    |   socket_send_line("grind_ready=True")
    | end
    | 
    | # Get into contact with part (or away from it)
    | # enable:  0=No Contact   1=Touch but no tool/coolant on or force  2=Touch, Tool, Coolant, and Force
    | def contact_part(on = False, enable = 0):
    |   if on:
    |     if enable == 0:
    |       # Just do a small forward motion in the direction of touchoff- this is a simulated p_contact_init
    |       global p_contact_init = pose_trans(iget_actual_tcp_pose(), p[0, 0, 0.005, 0, 0, 0])
    |       imovel(p_contact_init, a = robot_linear_accel_mpss, v = robot_linear_speed_mps)
    |     elif enable == 1:
    |       # Advance until contact but retract 2X grind distance and use this as a simulated p_contact_init
    |       local success = itouchoff(grind_touch_speed_mmps, grind_touch_retract_mm * 2.0)
    |       global p_contact_init = iget_actual_tcp_pose()
    |       return success
    |     elif enable == 2:
    |       # Advance until contact
    |       local success = itouchoff(grind_touch_speed_mmps, grind_touch_retract_mm)
    |       # Touchoff has backed off by grind_touch_retract_mm so we need to compute that actual p_contact_init
    |       global p_contact_init = pose_trans(iget_actual_tcp_pose(), p[0, 0, grind_touch_retract_mm / 1000.0, 0, 0, 0])
    |       return success
    |     end
    |   else:  # Back off
    |     local p1 = pose_trans(iget_actual_tcp_pose(), p[0, 0, -0.010, 0, 0, 0])
    |     imovel(p1, a = robot_linear_accel_mpss, v = robot_linear_speed_mps)
    |   end
    | 
    |   return True
    | end
    | 
    | # Sets digital outpus based 8-element list of 4 pairs DOUT#,State.  -1 indicates unused slot
    | def set_digital_output_list(list):
    |   i = 0
    |   while i < 8:
    |     if list[i] >= 0:
    |       b = list[i + 1] == 1
    |       set_digital_out(list[i], b)
    |     end
    |     i = i + 2
    |   end
    | end
    | 
    | # Turn tool power on/off if enable=2
    | def tool_power(on = False, enable = 0):
    |   if enable < 2:
    |     return None
    |   end
    | 
    |   if on:
    |     # ON IO
    |     set_digital_output_list(robot_tool_on_outputs)
    |   else:
    |     # OFF IO
    |     set_digital_output_list(robot_tool_off_outputs)
    |   end
    | 
    |   return None
    | end
    | 
    | # Turn coolant on/off if enable=2
    | def coolant_flow(on = False, enable = 0):
    |   if enable < 2:
    |     return None
    |   end
    | 
    |   if on:
    |     # ON IO
    |     set_digital_output_list(robot_coolant_on_outputs)
    |   else:
    |     # OFF IO
    |     set_digital_output_list(robot_coolant_off_outputs)
    |   end
    | 
    |   return None
    | end
    | 
    | # Turn force mode on/off if enable=2
    | def apply_force(on = False, enable = 0, force_n = 5, approach_speed_mmps = 10):
    |   if enable < 2:
    |     return None
    |   end
    | 
    |   if on:
    |     iforce_mode(force_n, approach_speed_mmps)
    |     sleep(grind_force_dwell_ms / 1000.0)
    |   else:
    |     iend_force_mode()
    |     sleep(0.1)
    |   end
    | 
    |   return None
    | end
    | 
    | # Update force applied only
    | def update_force(on = False, enable = 0, force_n = 5, approach_speed_mmps = 10):
    |   if enable < 2:
    |     return None
    |   end
    | 
    |   if on:
    |     iforce_update(force_n, approach_speed_mmps)
    |   end
    | 
    |   return None
    | end
    | 
    | # Start/Stop Grinding
    | # Pose to center is the offset we should move to initial touch point [0]=FLAT [1]=CYLINDER [2]=SPHERE
    | global grind_process_state = False
    | def set_grind_process_state(on = False, pose_to_center = [p[0, 0, 0, 0, 0, 0], p[0, 0, 0, 0, 0, 0], p[0, 0, 0, 0, 0, 0]]):
    |   if on and grind_process_state:
    |     # Continuing a grind...
    |     # Move to initial grind position relative to initial p_contact_center
    |     shape = robot_part_geometry[0]
    |     if shape < 1 or shape > 3:
    |       return False
    |     end
    |     global dp_from_contact_center = pose_to_center[shape-1]
    |     grind_to(dp_from_contact_center, r = 0)
    | 
    |     update_force(True, grind_contact_enable, grind_force_n, grind_touch_speed_mmps)
    |   elif on and not grind_process_state:
    |     # Need to start the grind
    |     global p_operator_init = iget_actual_tcp_pose()
    | 
    |     # Move to start position for touchoff
    |     shape = robot_part_geometry[0]
    |     if shape < 1 or shape > 3:
    |       return False
    |     end
    | 
    |     global dp_from_contact_center = pose_to_center[shape-1]
    |     local p1 = pose_trans(p_operator_init, dp_from_contact_center)
    |     # TODO This should look at whether rot or linear for speed,accel
    |     imovel(p1, a = robot_linear_accel_mpss, v = robot_linear_speed_mps)
    | 
    |     # Touch part and set p_contact_init
    |     if not contact_part(True, grind_contact_enable):
    |       # Failure to contact part should abort... don't set grind_process_state and return False
    |       imovel(p_operator_init, a = robot_linear_accel_mpss, v = robot_linear_speed_mps)
    |       socket_send_line("grind_process_state=False")
    |       return False
    |     end
    | 
    |     # Compute p_contact_center... where we would have been if we had touched off from the operator teach position!
    |     local  reverse_pose_to_center = pose_to_center[shape-1]
    |     local i = 0
    |     while i < 6:
    |       reverse_pose_to_center[i] = -reverse_pose_to_center[i]
    |       i = i + 1
    |     end
    |     global p_contact_center = pose_trans(p_contact_init, reverse_pose_to_center)
    |     grind_start(dp_from_contact_center)
    | 
    |     # Now power everything on (although these will do nothing unless contact_enable==2)
    |     tool_power(True, grind_contact_enable)
    |     coolant_flow(True, grind_contact_enable)
    |     apply_force(True, grind_contact_enable, grind_force_n, grind_touch_speed_mmps)
    |     global grind_process_state = True
    |   elif not on and grind_process_state:
    |     # Need to stop the grind
    |     # Shut everything down and return to original pose
    |     apply_force(False, grind_contact_enable, 0)
    |     contact_part(False, grind_contact_enable)
    |     coolant_flow(False, grind_contact_enable)
    |     tool_power(False, grind_contact_enable)
    |     imovel(p_operator_init, a = robot_linear_accel_mpss, v = robot_linear_speed_mps)
    |     global grind_process_state = False
    |   end
    | 
    |   # Always let the host know status
    |   if grind_process_state:
    |     socket_send_line("grind_process_state=True")
    |   else:
    |     socket_send_line("grind_process_state=False")
    |   end
    |   return True
    | end
    | 
    | ######################################################################################
    | # Thread to listen for abort messages while grinding
    | #
    | global grind_force_report_counter = 0
    | global grind_force_report = p[0, 0, 0, 0, 0, 0]
    | global grind_force_report_z_n = 0
    | thread grind_abort_listener_thread():
    |   global halt_command = [0, 0, 0, 0]
    |   global halt_count = 0
    |   global grind_force_report_counter = 0
    |   global grind_force_readings_n = 5
    |   global grind_force_readings = [0., 0., 0., 0., 0.]
    | 
    |   # Initialize force readings array
    |   local i = 0
    |   while i < grind_force_readings_n:
    |     local f = get_tcp_force()
    |     grind_force_readings[i] = f[2]
    |     i = i + 1
    |   end
    |   global grind_force_report_z_n = grind_force_readings[grind_force_readings_n-1]
    |   global grind_force_filtered_z_n = grind_force_report_z_n
    | 
    | 
    |   while (halt_count == 0):
    |     # Commands should never arrive, so this will block us for 0.2s
    |     global halt_command = socket_read_ascii_float(3, timeout = 0.2)
    | 
    |     # If door is open, that adds a halt count (anything >0 will stop us!)
    |     if not is_door_closed():
    |       global halt_count = halt_count + 1
    |     end
    | 
    |     # If we've received(index,checksum,10,...) that adds a halt count (as long as checksum matches)
    |     if halt_command[0] > 2:
    |       global test_index = halt_command[1]
    |       global test_checksum = halt_command[2]
    |       global test_command = halt_command[3]
    | 
    |       if test_checksum == 1000 - test_index and test_command == 10:
    |         global halt_count = halt_count + 1
    | 
    |         # Send an start/finish acknowledgement just for this command!
    |         socket_set_var("robot_starting", test_index)
    |         socket_set_var("robot_completed", test_index)
    |       end
    |     end
    | 
    |     # Increment reading counter (10000 is high enough... don't need to worry about wraparound effects)
    |     grind_force_report_counter = grind_force_report_counter + 1
    |     if grind_force_report_counter > 10000:
    |       grind_force_report_counter = 0
    |     end
    | 
    |     # Store force in circular buffer
    |     local force = get_tcp_force()
    |     grind_force_readings[grind_force_report_counter % grind_force_readings_n] = force[2]
    | 
    |     # Report force periodically (This executes at 5Hz because of timeout=0.2 in socket_read_ascii_float(...)
    |     if grind_force_report_counter % 5 == 0:
    |       # Compute average of the stored readings
    |       local i = 0
    |       local sum = 0.0
    |       while i < grind_force_readings_n:
    |         sum = sum + grind_force_readings[i]
    |         i = i + 1
    |       end
    |       global grind_force_average_z_n = sum / grind_force_readings_n
    | 
    |       # Any other filtering could be done here...
    |       # Round to 2 DP
    |       global grind_force_report_z_n = ceil(grind_force_average_z_n*100)/100
    | 
    |       socket_send_string("grind_force_report_z_n=")
    |       socket_send_string(grind_force_report_z_n)
    |       socket_send_lf()
    |     end
    |   end
    |   return None
    | end
    | 
    | # Should we proceed? halt_count==0 means no door-opens and no abort commands from host
    | def ok_to_proceed():
    |   return halt_count == 0
    | end
    | #
    | # Thread to listen for abort messages while grinding
    | ######################################################################################
    | 
    | 
    | ######################################################################################
    | # TOP LEVEL GRIND FUNCTIONS
    | #
    | # Grind along a line dx_mm x dy_mm centered on current tool position. Repeat n_cycles times. If stay_in_contact, stay_in_contact at end.
    | def grind_line(dx_mm, dy_mm, n_cycles, stay_in_contact):
    |   if n_cycles < 1:
    |     return True
    |   end
    | 
    |   # Unit conversion
    |   dx_m = dx_mm / 1000.0
    |   dy_m = dy_mm / 1000.0
    |   radius_m = robot_part_geometry[1] / 2000.0
    |   drx_rad = dx_m / radius_m
    |   dry_rad = dy_m / radius_m
    | 
    |   # Grind time estimate
    |   time_ms = sqrt(dx_mm * dx_mm + dy_mm * dy_mm) * n_cycles / grind_speed_mps + 1500
    |   socket_set_var("robot_step_time_estimate_ms", time_ms)
    | 
    |   # Swapping sphere axes here since RY is aligned with the X of the FLAT and CYLINDER geometries
    |   if not set_grind_process_state(True,
    |     [
    |       p[-dx_m / 2.0, -dy_m / 2.0, 0, 0, 0, 0],
    |       p[-dx_m / 2.0, 0, 0, -dry_rad / 2.0, 0, 0],
    |       p[0, 0, 0, -dry_rad / 2.0, -drx_rad / 2.0, 0]
    |     ]):
    |     return False
    |   end
    | 
    |   # Grind the pattern
    |   shape = robot_part_geometry[0]
    |   if shape == 1:
    |     pattern_line_flat(dx_m, dy_m, n_cycles)
    |   elif shape == 2:
    |     pattern_line_cylinder(dx_m, dry_rad, n_cycles)
    |   elif shape == 3:
    |     # Swapping axes here since RY is aligned with the X of the FLAT and CYLINDER geometries
    |     pattern_line_sphere(dry_rad, drx_rad, n_cycles)
    |   end
    | 
    |   if not stay_in_contact or not ok_to_proceed():
    |     set_grind_process_state(False)
    |   end
    |   return True
    | end
    | 
    | # Grind along a rect dx_mm x dy_mm centered on current tool position. Repeat n_cycles times. If stay_in_contact, stay_in_contact at end.
    | # Move in x direction first, then y
    | def grind_rect(dx_mm, dy_mm, n_cycles, stay_in_contact):
    |   if n_cycles < 1:
    |     return True
    |   end
    | 
    |   # Unit conversion
    |   dx_m = dx_mm / 1000.0
    |   dy_m = dy_mm / 1000.0
    |   diam_m = robot_part_geometry[1] / 1000.0
    |   radius_m = diam_m / 2.0
    |   drx_rad = dx_m / radius_m
    |   dry_rad = dy_m / radius_m
    | 
    |   # Grind time estimate
    |   time_ms = 2 * (dx_mm + dy_mm) * n_cycles / grind_speed_mps + 1500
    |   socket_set_var("robot_step_time_estimate_ms", time_ms)
    | 
    |   # Swapping sphere axes here since RY is aligned with the X of the FLAT and CYLINDER geometries
    |   # 4-point Version
    |   #if not set_grind_process_state(True,
    |   #  [
    |   #    p[-dx_m / 2.0, -dy_m / 2.0, 0, 0, 0, 0],
    |   #    p[-dx_m / 2.0, 0, 0, -dry_rad / 2.0, 0, 0],
    |   #    p[0, 0, 0, -dry_rad / 2.0, -drx_rad / 2.0, 0]
    |   #  ]):
    |   #  return False
    |   #end
    | 
    |   # 8-point Version
    |   if not set_grind_process_state(True,
    |     [
    |       p[-dx_m / 2.0 + grind_blend_radius_m * 2, -dy_m / 2.0, 0, 0, 0, 0],
    |       p[-dx_m / 2.0 + grind_blend_radius_m * 2, 0, 0, -dry_rad / 2.0, 0, 0],
    |       p[0, 0, 0, -dry_rad / 2.0 + grind_rot_blend_radius_rad * 8, -drx_rad / 2.0, 0]
    |     ]):
    |     return False
    |   end
    | 
    |   # Grind the pattern
    |   shape = robot_part_geometry[0]
    |   if shape == 1:
    |     pattern_rect_flat(dx_m, dy_m, n_cycles)
    |   elif shape == 2:
    |     pattern_rect_cylinder(dx_m, dry_rad, n_cycles)
    |   elif shape == 3:
    |     # Swapping sphere axes here since RY is aligned with the X of the FLAT and CYLINDER geometries
    |     pattern_rect_sphere(dry_rad, drx_rad, n_cycles)
    |   end
    | 
    |   if not stay_in_contact or not ok_to_proceed():
    |     set_grind_process_state(False)
    |   end
    |   return True
    | end
    | 
    | # Grind along a rect in serpentine dx_mm,dy_mm incrementing by xstep_mm,ystep_mm centered on current tool position. Repeat n_cycles times. If stay_in_contact, stay_in_contact at end.
    | # Move in x direction first, then y
    | def grind_serpentine(dx_mm, dy_mm, n_xsteps, n_ysteps, n_cycles, stay_in_contact):
    |   if n_cycles < 1:
    |     return True
    |   end
    | 
    |   # Either n_xsteps or n_ysteps must be 1. Whichever one is one will be the direction of the first move.
    |   if n_xsteps != 1 and n_ysteps != 1:
    |     return False
    |   end
    | 
    |   # Unit conversion
    |   dx_m = dx_mm / 1000.0
    |   dy_m = dy_mm / 1000.0
    |   part_radius_m = robot_part_geometry[1] / 2000.0
    |   drx_rad = dx_m / part_radius_m
    |   dry_rad = dy_m / part_radius_m
    | 
    |   # Grind time estimate
    |   # Per Cycle:
    |   # 1,3 does 4 passes in x and 1 in y     3,1 does 4 passes in Y and 1 in X
    |   #   ########################            #  ####  #
    |   #                          #            #  #  #  #
    |   #   ########################            #  #  #  #
    |   #   #                                   #  #  #  #
    |   #   ########################            #  #  #  #
    |   #                          #            #  #  #  #
    |   #   ########################            ####  ####
    |   if n_xsteps == 1:
    |     time_ms = (dx_mm * (n_ysteps + 1) + dy_mm) * n_cycles / grind_speed_mps + 1500
    |   else:
    |     time_ms = (dx_mm + dy_mm * (n_xsteps + 1)) * n_cycles / grind_speed_mps + 1500
    |   end
    |   socket_set_var("robot_step_time_estimate_ms", time_ms)
    | 
    |   # Swapping sphere axes here since RY is aligned with the X of the FLAT and CYLINDER geometries
    |   if not set_grind_process_state(True,
    |     [
    |       p[-dx_m / 2.0, -dy_m / 2.0, 0, 0, 0, 0],
    |       p[-dx_m / 2.0, 0, 0, -dry_rad / 2.0, 0, 0],
    |       p[0, 0, 0, -dry_rad / 2.0, -drx_rad / 2.0, 0]
    |     ]):
    |     return False
    |   end
    | 
    |   # Grind the pattern
    |   shape = robot_part_geometry[0]
    |   if shape == 1:
    |     pattern_serpentine_flat(dx_m, dy_m, n_xsteps, n_ysteps, n_cycles)
    |   elif shape == 2:
    |     pattern_serpentine_cylinder(dx_m, dry_rad, n_xsteps, n_ysteps, n_cycles)
    |   elif shape == 3:
    |     # Swapping axes here since RY is aligned with the X of the FLAT and CYLINDER geometries
    |     pattern_serpentine_sphere(dry_rad, drx_rad, n_ysteps, n_xsteps, n_cycles)
    |   end
    | 
    |   if not stay_in_contact or not ok_to_proceed():
    |     set_grind_process_state(False)
    |   end
    |   return True
    | end
    | 
    | # Grind along a polygon with circle_diam_mm and n_sides. Repeat n_cycles times. If stay_in_contact, stay_in_contact at end.
    | def grind_poly(circle_diam_mm, n_sides, n_cycles, stay_in_contact):
    |   if n_cycles < 1:
    |     return True
    |   end
    | 
    |   # Unit conversion
    |   local circle_diam_m = circle_diam_mm / 1000.0
    |   local part_diam_m = robot_part_geometry[1] / 1000.0
    | 
    |   # Grind time estimate
    |   local time_ms = MATH_PI * circle_diam_mm * n_cycles / grind_speed_mps + 1500
    |   socket_set_var("robot_step_time_estimate_ms", time_ms)
    | 
    |   if not set_grind_process_state(True,
    |     [
    |       p[-circle_diam_m / 2.0, 0, 0, 0, 0, 0],
    |       p[-circle_diam_m / 2.0, 0, 0, 0, 0, 0],
    |       p[0, 0, 0, -circle_diam_m / part_diam_m, 0, 0]
    |     ]):
    |     return False
    |   end
    | 
    |   # Grind the pattern
    |   local shape = robot_part_geometry[0]
    |   if shape == 1:
    |     pattern_poly_flat(circle_diam_m, n_sides, n_cycles)
    |   elif shape == 2:
    |     pattern_poly_cylinder(circle_diam_m, n_sides, part_diam_m, n_cycles)
    |   elif shape == 3:
    |     pattern_poly_sphere(circle_diam_m, n_sides, part_diam_m, n_cycles)
    |   end
    | 
    |   if not stay_in_contact or not ok_to_proceed():
    |     set_grind_process_state(False)
    |   end
    |   return True
    | end
    | 
    | def recommend_npoints(diam_m):
    |   # 1 point per second?
    |   local circum_m = MATH_PI * diam_m
    |   local t = circum_m / grind_speed_mps
    |   global grind_circle_n_sides = limiter(ceil(t * 2), 2, 1000)
    | 
    |   # 100mm diam gets 50 points... seems about right
    |   #global grind_circle_n_sides = limiter(diam_m * 500, 2, 1000)
    |   return grind_circle_n_sides
    | end
    | 
    | # Grind along a circle with circle_diam_mm. Repeat n_cycles times. If stay_in_contact, stay_in_contact at end.
    | def grind_circle(circle_diam_mm, n_cycles, stay_in_contact):
    |   global grind_circle_n_sides = recommend_npoints(circle_diam_mm / 1000.0)
    | 
    |   if grind_blend_radius_m > 0.0:
    |     # Try setting n_sides to 1.5 blend radii
    |     local circum_m = MATH_PI * circle_diam_mm / 1000.
    |     global grind_circle_n_sides = ceil(circum_m / (grind_blend_radius_m * 1.5))
    |   end
    |   return grind_poly(circle_diam_mm, grind_circle_n_sides, n_cycles, stay_in_contact)
    | end
    | 
    | # Grind along a spiral circle1_diam_mm to circle2_diam_mm in n_revolutions with rotations centered on current tool position. Repeat n_cycles times. If stay_in_contact, stay_in_contact at end.
    | def grind_spiral(circle1_diam_mm, circle2_diam_mm, n_revolutions, n_cycles, stay_in_contact):
    |   if n_cycles < 1:
    |     return True
    |   end
    | 
    |   # Unit conversion
    |   local circle1_diam_m = circle1_diam_mm / 1000.0
    |   local circle2_diam_m = circle2_diam_mm / 1000.0
    |   local part_diam_m = robot_part_geometry[1] / 1000.0
    | 
    |   # Grind time estimate based on average diam
    |   local avg_diam_mm = (circle1_diam_mm + circle2_diam_mm) / 2.0
    |   local time_ms = MATH_PI * avg_diam_mm * n_revolutions * n_cycles / grind_speed_mps + 1500
    |   socket_set_var("robot_step_time_estimate_ms", time_ms)
    | 
    |   if not set_grind_process_state(True,
    |     [
    |       p[-circle1_diam_m / 2.0, 0, 0, 0, 0, 0],
    |       p[-circle1_diam_m / 2.0, 0, 0, 0, 0, 0],
    |       p[0, 0, 0, -circle1_diam_m / part_diam_m, 0, 0]
    |     ]):
    |     return False
    |   end
    | 
    |   # Grind the pattern
    |   local shape = robot_part_geometry[0]
    |   if shape == 1:
    |     pattern_spiral_flat(circle1_diam_m, circle2_diam_m, n_revolutions, n_cycles)
    |   elif shape == 2:
    |     pattern_spiral_cylinder(circle1_diam_m, circle2_diam_m, n_revolutions, part_diam_m, n_cycles)
    |   elif shape == 3:
    |     pattern_spiral_sphere(circle1_diam_m, circle2_diam_m, n_revolutions, part_diam_m, n_cycles)
    |   end
    | 
    |   if not stay_in_contact or not ok_to_proceed():
    |     set_grind_process_state(False)
    |   end
    |   return True
    | end
    | 
    | 
    | ######################################################################################
    | ######################################################################################
    | #
    | # PATTERN GRINDING FUNCTIONS
    | #
    | global grind_current_dp = p[0, 0, 0, 0, 0, 0]
    | 
    | def grind_start(current_dp):
    |   global grind_current_dp = p[0, 0, 0, 0, 0, 0]
    | 
    |   grind_to(current_dp)
    | end
    | 
    | def grind_to(dp, r = -1, no_wait = False):
    |   global grind_current_ddp0 = abs(dp[0] - grind_current_dp[0])
    |   global grind_current_ddp1 = abs(dp[1] - grind_current_dp[1])
    |   global grind_current_ddp3 = abs(dp[3] - grind_current_dp[3])
    |   global grind_current_ddp4 = abs(dp[4] - grind_current_dp[4])
    |   # Flat:     X, Y
    |   # Cylinder: X, RX
    |   # Sphere:   RX, RX
    |   local shape = robot_part_geometry[0]
    |   if shape == 3: # Sphere
    |     global process_a = grind_rot_accel_rpss
    |     global process_v = grind_rot_speed_rps
    |     global process_r = grind_rot_blend_radius_rad
    |   elif shape == 2: # Cylinder
    |     global process_theta = atan2(grind_current_ddp3, grind_current_ddp0)
    |     global process_rotational_factor = abs(sin(process_theta))
    |     global process_a =
    |     (
    |       grind_accel_mpss * (1 - process_rotational_factor) +
    |       grind_rot_accel_rpss * (process_rotational_factor)
    |     )
    |     global process_v =
    |     (
    |       grind_speed_mps * (1 - process_rotational_factor) +
    |       grind_rot_speed_rps * (process_rotational_factor)
    |     )
    |     global process_r =
    |     (
    |       grind_blend_radius_m * (1 - process_rotational_factor) +
    |       grind_rot_blend_radius_rad * (process_rotational_factor)
    |     )
    |   else: # Flat
    |     global process_a = grind_accel_mpss
    |     global process_v = grind_speed_mps
    |     global process_r = grind_blend_radius_m
    |   end
    | 
    |   global process_r_in = r
    |   if r >= 0:
    |     global process_r = r
    |   end
    | 
    |   global grind_current_dp = dp
    |   imovel_int(pose_trans(p_contact_center, grind_current_dp), a = process_a, v = process_v, r = process_r, no_wait = no_wait)
    | end
    | 
    | def grind_finish(p):
    |   grind_to(p, r = 0)
    | end
    | 
    | ######################################################################################
    | # LINE PATTERNS
    | #
    | # The line pattern sequence.
    | # Assumes all point_dist are declared globally
    | def pattern_line(n_cycles):
    |   global grind_cycle = 1
    |   local dpdest = dp2
    |   while (ok_to_proceed() and grind_cycle <= n_cycles):
    |     socket_set_var("grind_cycle", grind_cycle)
    | 
    |     if grind_cycle == n_cycles:
    |       grind_finish(dpdest)
    |     else:
    |       grind_to(dpdest, r = 0)
    |     end
    | 
    |     if dpdest == dp1:
    |       dpdest = dp2
    |     else:
    |       dpdest = dp1
    |     end
    | 
    |     grind_cycle = grind_cycle + 1
    |   end
    | end
    | 
    | # Move along a flat line dx_m x dy_m. Repeat n_cycles times.
    | # Move in x direction first, then y
    | def pattern_line_flat(dx_m, dy_m, n_cycles):
    |   local x2 = dx_m / 2.0
    |   local y2 = dy_m / 2.0
    | 
    |   global dp1 = dp_from_contact_center
    |   global dp2 = p[x2, y2, 0, 0, 0, 0]
    | 
    |   pattern_line(n_cycles)
    | end
    | 
    | # Move along a cylindrical line dx_m x dy_m. Repeat n_cycles times.
    | # Move in x direction first, then y
    | def pattern_line_cylinder(dx_m, drx_rad, n_cycles):
    |   local x2 = dx_m / 2.0
    |   local rx2 = drx_rad / 2.0
    | 
    |   global dp1 = dp_from_contact_center
    |   global dp2 = p[x2, 0, 0, rx2, 0, 0]
    | 
    |   pattern_line(n_cycles)
    | end
    | 
    | # Move along a sphere line dx_m x dy_m. Repeat n_cycles times.
    | # Move in x direction first, then y
    | def pattern_line_sphere(drx_rad, dry_rad, n_cycles):
    |   local rx2 = drx_rad / 2.0
    |   local ry2 = dry_rad / 2.0
    | 
    |   global dp1 = dp_from_contact_center
    |   global dp2 = p[0, 0, 0, rx2, ry2, 0]
    | 
    |   pattern_line(n_cycles)
    | end
    | 
    | ######################################################################################
    | # RECT PATTERNS
    | #
    | # The rect pattern sequence. Assumes all points are defined globally!
    | def pattern_rect(n_cycles):
    |   global grind_cycle = 1
    |   while (ok_to_proceed() and grind_cycle <= n_cycles):
    |     socket_set_var("grind_cycle", grind_cycle)
    | 
    |     # 4-point Version
    |     #grind_finish(dp2)
    |     #grind_finish(dp3)
    |     #grind_finish(dp4)
    |     #grind_finish(dp1)
    | 
    |     # 8-point Version
    |     grind_finish(dp2a)
    |     grind_finish(dp2b)
    |     grind_finish(dp3a)
    |     grind_finish(dp3b)
    |     grind_finish(dp4a)
    |     grind_finish(dp4b)
    |     grind_finish(dp1a)
    |     grind_finish(dp1b)
    | 
    |     grind_cycle = grind_cycle + 1
    |   end
    | end
    | 
    | # Move along a flat rect dx_m x dy_m. Repeat n_cycles times.
    | # Move in x direction first, then y
    | def pattern_rect_flat(dx_m, dy_m, n_cycles):
    |   local x2 = dx_m / 2.0
    |   local y2 = dy_m / 2.0
    | 
    |   local dx = grind_blend_radius_m * 2
    | 
    |   global dp1 = p[-x2, -y2, 0, 0, 0, 0]
    |   global dp1a = dp1
    |   global dp1b = dp1
    |   dp1a[1] = dp1a[1] + dx
    |   dp1b[0] = dp1b[0] + dx
    | 
    |   global dp2 = p[x2, -y2, 0, 0, 0, 0]
    |   global dp2a = dp2
    |   global dp2b = dp2
    |   dp2a[0] = dp2a[0] - dx
    |   dp2b[1] = dp2b[1] + dx
    | 
    |   global dp3 = p[x2, y2, 0, 0, 0, 0]
    |   global dp3a = dp3
    |   global dp3b = dp3
    |   dp3a[1] = dp3a[1] - dx
    |   dp3b[0] = dp3b[0] - dx
    | 
    |   global dp4 = p[-x2, y2, 0, 0, 0, 0]
    |   global dp4a = dp4
    |   global dp4b = dp4
    |   dp4a[0] = dp4a[0] + dx
    |   dp4b[1] = dp4b[1] - dx
    | 
    |   pattern_rect(n_cycles)
    | end
    | 
    | # Move along a cylindrical rect dx_mm,drx_rad. Repeat n_cycles times.
    | # Move in x direction first, then rx
    | def pattern_rect_cylinder(dx_m, drx_rad, n_cycles):
    |   local x2 = dx_m / 2.0
    |   local rx2 = drx_rad / 2.0
    | 
    |   local dx = grind_blend_radius_m * 2
    |   local da = grind_rot_blend_radius_rad * 8
    | 
    |   global dp1 = p[-x2, 0, 0, -rx2, 0, 0]
    |   global dp1a = dp1
    |   global dp1b = dp1
    |   dp1a[3] = dp1a[3] + da
    |   dp1b[0] = dp1b[0] + dx
    | 
    |   global dp2 = p[x2, 0, 0, -rx2, 0, 0]
    |   global dp2a = dp2
    |   global dp2b = dp2
    |   dp2a[0] = dp2a[0] - dx
    |   dp2b[3] = dp2b[3] + da
    | 
    |   global dp3 = p[x2, 0, 0, rx2, 0, 0]
    |   global dp3a = dp3
    |   global dp3b = dp3
    |   dp3a[3] = dp3a[3] - da
    |   dp3b[0] = dp3b[0] - dx
    | 
    |   global dp4 = p[-x2, 0, 0, rx2, 0, 0]
    |   global dp4a = dp4
    |   global dp4b = dp4
    |   dp4a[0] = dp4a[0] + dx
    |   dp4b[3] = dp4b[3] - da
    | 
    |   pattern_rect(n_cycles)
    | end
    | 
    | # Move along a spherical rect drx_rad,dry_rad. Repeat n_cycles times.
    | # Move in rx direction first, then ry
    | def pattern_rect_sphere(drx_rad, dry_rad, n_cycles):
    |   local rx2 = drx_rad / 2.0
    |   local ry2 = dry_rad / 2.0
    | 
    |   local da = grind_rot_blend_radius_rad * 8
    | 
    |   global dp1 = p[0, 0, 0, -rx2, -ry2, 0]
    |   global dp1a = dp1
    |   global dp1b = dp1
    |   dp1a[4] = dp1a[4] + da
    |   dp1b[3] = dp1b[3] + da
    | 
    |   global dp2 = p[0, 0, 0, rx2, -ry2, 0]
    |   global dp2a = dp2
    |   global dp2b = dp2
    |   dp2a[3] = dp2a[3] - da
    |   dp2b[4] = dp2b[4] + da
    | 
    |   global dp3 = p[0, 0, 0, rx2, ry2, 0]
    |   global dp3a = dp3
    |   global dp3b = dp3
    |   dp3a[4] = dp3a[4] - da
    |   dp3b[3] = dp3b[3] - da
    | 
    |   global dp4 = p[0, 0, 0, -rx2, ry2, 0]
    |   global dp4a = dp4
    |   global dp4b = dp4
    |   dp4a[3] = dp4a[3] + da
    |   dp4b[4] = dp4b[4] - da
    | 
    |   pattern_rect(n_cycles)
    | end
    | 
    | ######################################################################################
    | # SERPENTINE PATTERNS
    | #
    | # Move along a flat serpentine dx_m,dy_m in n_xsteps,n_ysteps. Repeat n_cycles times.
    | # Move in direction of whichever nsteps is 1 first
    | def pattern_serpentine_flat(dx_m, dy_m, n_xsteps, n_ysteps, n_cycles):
    |   local t_move_x = dx_m / grind_speed_mps
    |   local t_move_y = dy_m / grind_speed_mps
    | 
    |   # Bottom left corner, grid 0,0
    |   local x2 = dx_m / 2.0
    |   local y2 = dy_m / 2.0
    |   local dp1 = dp_from_contact_center
    |   local dp2 = dp1
    | 
    |   # Track our grid square number... we're in [0,0] and moving [+1,+1] in either x or y
    |   local x_grid = 0
    |   local y_grid = 0
    |   local x_incr = 1
    |   local y_incr = 1
    |   local grid_dx_m = dx_m / n_xsteps
    |   local grid_dy_m = dy_m / n_ysteps
    | 
    |   # How many moves does it take to complete a pass?
    |   global n_moves_per_pass = (n_xsteps + n_ysteps) * 2 - 1
    | 
    |   local move_count = 0
    |   global grind_cycle = 1
    |   while (ok_to_proceed() and grind_cycle <= n_cycles):
    |     # This will repeat for each leg of the serpentine!
    |     socket_set_var("grind_cycle", grind_cycle)
    | 
    |     # Skip first X move if we should start with a y move
    |     if move_count != 0 or n_xsteps == 1:
    |       # Advance x_grid by x_incr
    |       x_grid = x_grid + x_incr
    | 
    |       # Move to the corresponding position
    |       local dp2 = p[x_grid * grid_dx_m - x2, y_grid * grid_dy_m - y2, 0, 0, 0, 0]
    |       grind_finish(dp2)
    | 
    |       # Adjust x direction
    |       if x_grid >= n_xsteps:
    |         x_incr = -1
    |       elif x_grid <= 0:
    |         x_incr = 1
    |       end
    |       move_count = move_count + 1
    |     end
    | 
    |     if ok_to_proceed() and move_count < n_moves_per_pass:
    |       # Advance y_grid by y_incr
    |       y_grid = y_grid + y_incr
    | 
    |       # Move to the corresponding position
    |       local dp2 = p[x_grid * grid_dx_m - x2, y_grid * grid_dy_m - y2, 0, 0, 0, 0]
    |       grind_finish(dp2)
    | 
    |       # Adjust y direction
    |       if y_grid >= n_ysteps:
    |         y_incr = -1
    |       elif y_grid <= 0:
    |         y_incr = 1
    |       end
    |       move_count = move_count + 1
    |     end
    | 
    |     # Detect when we've covered all the grid squares!
    |     if move_count >= n_moves_per_pass:
    |       grind_cycle = grind_cycle + 1
    |       move_count = 0
    |     end
    |   end
    | end
    | 
    | # Move along a cylindrical serpentine dx_m,drx_rad in n_xsteps,n_rxsteps. Repeat n_cycles times.
    | # Move in direction of whichever nsteps is 1 first
    | def pattern_serpentine_cylinder(dx_m, drx_rad, n_xsteps, n_rxsteps, n_cycles):
    |   local t_move_x = dx_m / grind_speed_mps
    |   local t_move_rx = drx_rad / grind_rot_speed_rps / 4
    | 
    |   # Bottom left corner, grid 0,0
    |   local x2 = dx_m / 2.0
    |   local rx2 = drx_rad / 2.0
    |   local dp1 = dp_from_contact_center
    |   local dp2 = dp1
    | 
    |   # Track our grid square number... we're in [0,0] and moving [+1,+1] in either x or y
    |   local x_grid = 0
    |   local y_grid = 0
    |   local x_incr = 1
    |   local y_incr = 1
    |   local grid_dx_m = dx_m / n_xsteps
    |   local grid_drx_rad = drx_rad / n_rxsteps
    |   local last_a = grind_accel_mpss
    |   local last_v = grind_speed_mps
    | 
    |   # How many moves does it take to complete a pass?
    |   global n_moves_per_pass = (n_xsteps + n_rxsteps) * 2 - 1
    | 
    |   local move_count = 0
    |   global grind_cycle = 1
    |   grind_start(dp1)
    |   while (ok_to_proceed() and grind_cycle <= n_cycles):
    |     # This will repeat for each leg of the serpentine!
    |     socket_set_var("grind_cycle", grind_cycle)
    | 
    |     # Skip first X move if we should start with a y move
    |     if move_count != 0 or n_xsteps == 1:
    |       # Advance x_grid by x_incr
    |       x_grid = x_grid + x_incr
    | 
    |       # Move to the corresponding position
    |       local dp2 = p[x_grid * grid_dx_m - x2, 0, 0, y_grid * grid_drx_rad - rx2, 0, 0]
    |       local last_a = grind_accel_mpss
    |       local last_v = grind_speed_mps
    |       grind_finish(dp2)
    | 
    |       # Adjust x direction
    |       if x_grid >= n_xsteps:
    |         x_incr = -1
    |       elif x_grid <= 0:
    |         x_incr = 1
    |       end
    |       move_count = move_count + 1
    |     end
    | 
    |     if ok_to_proceed() and move_count < n_moves_per_pass:
    |       # Advance y_grid by y_incr
    |       y_grid = y_grid + y_incr
    | 
    |       # Move to the corresponding position
    |       local dp2 = p[x_grid * grid_dx_m - x2, 0, 0, y_grid * grid_drx_rad - rx2, 0, 0]
    |       local last_a = grind_rot_accel_rpss
    |       local last_v = grind_rot_speed_rps
    |       grind_finish(dp2)
    | 
    |       # Adjust y direction
    |       if y_grid >= n_rxsteps:
    |         y_incr = -1
    |       elif y_grid <= 0:
    |         y_incr = 1
    |       end
    |       move_count = move_count + 1
    |     end
    | 
    |     # Detect when we've covered all the grid squares!
    |     if move_count >= n_moves_per_pass:
    |       grind_cycle = grind_cycle + 1
    |       move_count = 0
    |     end
    |   end
    | end
    | 
    | # Move along a sperical serpentine drx_rad,dry_rad in n_rxsteps,n_rysteps. Repeat n_cycles times.
    | # Move in direction of whichever nsteps is 1 first
    | def pattern_serpentine_sphere(drx_rad, dry_rad, n_rxsteps, n_rysteps, n_cycles):
    |   local t_move_rx = drx_rad / grind_rot_speed_rps / 4
    |   local t_move_ry = dry_rad / grind_rot_speed_rps / 4
    | 
    |   # Bottom left corner, grid 0,0
    |   local rx2 = drx_rad / 2.0
    |   local ry2 = dry_rad / 2.0
    |   local dp1 = dp_from_contact_center
    |   local dp2 = dp1
    | 
    |   # Track our grid square number... we're in [0,0] and moving [+1,+1] in either x or y
    |   local x_grid = 0
    |   local y_grid = 0
    |   local x_incr = 1
    |   local y_incr = 1
    |   local grid_drx_rad = drx_rad / n_rxsteps
    |   local grid_dry_rad = dry_rad / n_rysteps
    | 
    |   # How many moves does it take to complete a pass?
    |   global n_moves_per_pass = (n_rxsteps + n_rysteps) * 2 - 1
    | 
    |   local move_count = 0
    |   global grind_cycle = 1
    |   grind_start(dp1)
    |   while (ok_to_proceed() and grind_cycle <= n_cycles):
    |     # This will repeat for each leg of the serpentine!
    |     socket_set_var("grind_cycle", grind_cycle)
    | 
    |     # Skip first X move if we should start with a y move
    |     if move_count != 0 or n_rxsteps == 1:
    |       # Advance x_grid by x_incr
    |       x_grid = x_grid + x_incr
    | 
    |       # Move to the corresponding position
    |       local dp2 = p[0, 0, 0, x_grid * grid_drx_rad - rx2, y_grid * grid_dry_rad - ry2, 0]
    |       grind_finish(dp2)
    | 
    |       # Adjust x direction
    |       if x_grid >= n_rxsteps:
    |         x_incr = -1
    |       elif x_grid <= 0:
    |         x_incr = 1
    |       end
    |       move_count = move_count + 1
    |     end
    | 
    |     if ok_to_proceed() and move_count < n_moves_per_pass:
    |       # Advance y_grid by y_incr
    |       y_grid = y_grid + y_incr
    | 
    |       # Move to the corresponding position
    |       local dp2 = p[0, 0, 0, x_grid * grid_drx_rad - rx2, y_grid * grid_dry_rad - ry2, 0]
    |       grind_finish(dp2)
    | 
    |       # Adjust y direction
    |       if y_grid >= n_rysteps:
    |         y_incr = -1
    |       elif y_grid <= 0:
    |         y_incr = 1
    |       end
    |       move_count = move_count + 1
    |     end
    | 
    |     # Detect when we've covered all the grid squares!
    |     if move_count >= n_moves_per_pass:
    |       grind_cycle = grind_cycle + 1
    |       move_count = 0
    |     end
    |   end
    | end
    | 
    | 
    | ######################################################################################
    | # POLYGONAL PATTERNS
    | #
    | # Grind along a polygon with circle_diam_m and n_sides on a flat. Repeat n_cycles times.
    | def pattern_poly_flat(circle_diam_m, n_sides, n_cycles):
    |   # Local calculations
    |   local circle_radius_m = circle_diam_m / 2.0
    | 
    |   global grind_cycle = 1
    |   while (ok_to_proceed() and grind_cycle <= n_cycles):
    |     socket_set_var("grind_cycle", grind_cycle)
    |     local i = 0
    |     while ok_to_proceed() and i <= n_sides:
    |       local theta = d2r(180.0 + 360.0 * i / n_sides)
    |       local x = circle_radius_m * cos(theta)
    |       local y = circle_radius_m * sin(theta)
    | 
    |       local dp = p[x, y, 0, 0, 0, 0]
    |       if not ok_to_proceed() or i == n_sides:
    |         grind_finish(dp)
    |       else:
    |         grind_to(dp)
    |       end
    |       i = i + 1
    |     end
    | 
    |     grind_cycle = grind_cycle + 1
    |   end
    | end
    | 
    | # Grind along a polygon with circle_diam_m and n_sides on a cylinder_radius_m. Repeat n_cycles times.
    | def pattern_poly_cylinder(circle_diam_m, n_sides, cylinder_radius_m, n_cycles):
    |   # Local calculations
    |   local circle_radius_m = circle_diam_m / 2.0
    | 
    |   global grind_cycle = 1
    |   while (ok_to_proceed() and grind_cycle <= n_cycles):
    |     socket_set_var("grind_cycle", grind_cycle)
    |     local i = 0
    |     while ok_to_proceed() and i <= n_sides:
    |       local theta = d2r(180.0 + 360.0 * i / n_sides)
    |       local x = circle_radius_m * cos(theta)
    |       local y = circle_radius_m * sin(theta)
    |       local rx = 2.0 * y / cylinder_radius_m
    | 
    |       local dp = p[x, 0, 0, rx, 0, 0]
    |       if not ok_to_proceed() or i == n_sides:
    |         grind_finish(dp)
    |       else:
    |         grind_to(dp)
    |       end
    |       i = i + 1
    |     end
    | 
    |     grind_cycle = grind_cycle + 1
    |   end
    | end
    | 
    | # Grind along a polygon with circle_diam_m and n_sides on a sphere_diam_m. Repeat n_cycles times.
    | def pattern_poly_sphere(circle_diam_m, n_sides, sphere_diam_m, n_cycles):
    |   # Local calculations
    |   local circle_radius_m = circle_diam_m / 2.0
    |   local sphere_radius_m = sphere_diam_m / 2.0
    | 
    |   global grind_cycle = 1
    |   while (ok_to_proceed() and grind_cycle <= n_cycles):
    |     socket_set_var("grind_cycle", grind_cycle)
    |     local i = 0
    |     while ok_to_proceed() and i <= n_sides:
    |       local theta = d2r(180.0 + 360.0 * i / n_sides)
    |       local x = circle_radius_m * cos(theta)
    |       local rx = x / sphere_radius_m
    |       local y = circle_radius_m * sin(theta)
    |       local ry = y / sphere_radius_m
    | 
    |       local dp = p[0, 0, 0, rx, ry, 0]
    |       if not ok_to_proceed() or i == n_sides:
    |         grind_finish(dp)
    |       else:
    |         grind_to(dp)
    |       end
    |       i = i + 1
    |     end
    | 
    |     grind_cycle = grind_cycle + 1
    |   end
    | end
    | 
    | 
    | ######################################################################################
    | # SPIRAL PATTERNS
    | #
    | # Grind a flat spiral from diam1 to diam2 in n_revolutions revolutions
    | def pattern_spiral_flat(circle1_diam_m, circle2_diam_m, n_revolutions, n_cycles):
    |   # Local calculations
    |   local max_diam_m = max(circle1_diam_m, circle2_diam_m)
    |   local n_points = recommend_npoints(max_diam_m)
    |   local n_total_points = n_revolutions * n_points
    |   local circle1_radius_m = circle1_diam_m / 2.0
    |   local circle2_radius_m = circle2_diam_m / 2.0
    | 
    |   global grind_cycle = 1
    |   while (ok_to_proceed() and grind_cycle <= n_cycles):
    |     socket_set_var("grind_cycle", grind_cycle)
    |     local rslope = (circle2_radius_m - circle1_radius_m) / n_total_points
    |     local i = 0
    |     while ok_to_proceed() and i <= n_total_points:
    |       local theta = d2r(180.0 + 360.0 * (i % n_points) / n_points)
    |       local r_instantaneous = i * rslope + circle1_radius_m
    |       local x = r_instantaneous * cos(theta)
    |       local y = r_instantaneous * sin(theta)
    | 
    |       local dp = p[x, y, 0, 0, 0, 0]
    |       if not ok_to_proceed() or i == n_points:
    |         grind_finish(dp)
    |       else:
    |         grind_to(dp)
    |       end
    |       i = i + 1
    |     end
    |     grind_cycle = grind_cycle + 1
    | 
    |     # Next cycle- swap diameters so we go in/out/in etc.
    |     local old_circle1_radius_m = circle1_radius_m
    |     local circle1_radius_m = circle2_radius_m
    |     local circle2_radius_m = old_circle1_radius_m
    |   end
    | end
    | 
    | # Grind a spiral on a cylinder from diam1 to diam2 in n_revolutions revolutions
    | def pattern_spiral_cylinder(circle1_diam_m, circle2_diam_m, n_revolutions, cylinder_radius_m, n_cycles):
    |   # Local calculations
    |   local max_diam_m = max(circle1_diam_m, circle2_diam_m)
    |   local n_points = recommend_npoints(max_diam_m)
    |   local n_total_points = n_revolutions * n_points
    |   local circle1_radius_m = circle1_diam_m / 2.0
    |   local circle2_radius_m = circle2_diam_m / 2.0
    | 
    |   global grind_cycle = 1
    |   while (ok_to_proceed() and grind_cycle <= n_cycles):
    |     socket_set_var("grind_cycle", grind_cycle)
    |     local rslope = (circle2_radius_m - circle1_radius_m) / n_total_points
    |     local i = 0
    |     while ok_to_proceed() and i <= n_total_points:
    |       local theta = d2r(180.0 + 360.0 * (i % n_points) / n_points)
    |       local r_instantaneous = i * rslope + circle1_radius_m
    |       local x = r_instantaneous * cos(theta)
    |       local y = r_instantaneous * sin(theta)
    |       local rx = 2.0 * y / cylinder_radius_m
    | 
    |       local dp = p[x, 0, 0, rx, 0, 0]
    | 
    |       if not ok_to_proceed() or i == n_points:
    |         grind_finish(dp)
    |       else:
    |         grind_to(dp)
    |       end
    |       i = i + 1
    |     end
    |     grind_cycle = grind_cycle + 1
    | 
    |     # Next cycle- swap diameters so we go in/out/in etc.
    |     local old_circle1_radius_m = circle1_radius_m
    |     local circle1_radius_m = circle2_radius_m
    |     local circle2_radius_m = old_circle1_radius_m
    |   end
    | end
    | 
    | # Grind a spiral on a sphere from diam1 to diam2 in n_revolutions revolutions
    | def pattern_spiral_sphere(circle1_diam_m, circle2_diam_m, n_revolutions, sphere_diam_m, n_cycles):
    |   # Local calculations
    |   local max_diam_m = max(circle1_diam_m, circle2_diam_m)
    |   local n_points = recommend_npoints(max_diam_m)
    |   local n_total_points = n_revolutions * n_points
    |   local circle1_radius_m = circle1_diam_m / 2.0
    |   local circle2_radius_m = circle2_diam_m / 2.0
    |   local sphere_radius_m = sphere_diam_m / 2.0
    | 
    |   global grind_cycle = 1
    |   while (ok_to_proceed() and grind_cycle <= n_cycles):
    |     socket_set_var("grind_cycle", grind_cycle)
    |     local rslope = (circle2_radius_m - circle1_radius_m) / n_total_points
    |     local i = 0
    |     while ok_to_proceed() and i <= n_total_points:
    |       local theta = d2r(180.0 + 360.0 * (i % n_points) / n_points)
    |       local r_instantaneous = i * rslope + circle1_radius_m
    |       local x = r_instantaneous * cos(theta)
    |       local rx = x / sphere_radius_m
    |       local y = r_instantaneous * sin(theta)
    |       local ry = y / sphere_radius_m
    | 
    |       local dp = p[0, 0, 0, rx, ry, 0]
    |       if not ok_to_proceed() or i == n_points:
    |         grind_finish(dp)
    |       else:
    |         grind_to(dp)
    |       end
    |       i = i + 1
    |     end
    |     grind_cycle = grind_cycle + 1
    | 
    |     # Next cycle- swap diameters so we go in/out/in etc.
    |     local old_circle1_radius_m = circle1_radius_m
    |     local circle1_radius_m = circle2_radius_m
    |     local circle2_radius_m = old_circle1_radius_m
    |   end
    | end
  currentTcpPose := get_actual_tcp_pose()
  MoveJ speed 60 deg/s, acceleration 80 deg/s^2 (useActiveTCP=true) feature=Base
    Waypoint Waypoint (Variable): variable=currentTcpPose
  socket_is_open := False
Robot Program (runOnlyOnce=false)
  Loop While (checkContinuously=false) expression=socket_is_open ≟  False
    Wait Sleep waitTime=0.25
    Script: socket_close()
    socket_is_open := socket_open("169.254.254.200", 30000)
    If not socket_is_open
      socket_is_open := socket_open("169.254.254.210", 30000)
    If not socket_is_open
      socket_is_open := socket_open("192.168.0.252", 30000)
  response := "Unknown command"
  command := socket_read_ascii_float(12)
  If command_validate()
    Script: command_start()
    Set DigitalOutput pin=Stacklight; digitalValue=1
    Switch expression=command[1]
      Case (caseValue=10)
        Script: return_actual_tcp_pose()
      Case (caseValue=12)
        Script: return_tcp_offset()
      Case (caseValue=13)
        Script: movel_relative_base(p[command[2], command[3], command[4], command[5], command[6], command[7]])
      Case (caseValue=14)
        Script: movel_relative_tcp(p[command[2], command[3], command[4], command[5], command[6], command[7]])
      Case (caseValue=15)
        Script: movel_relative_tcp_part(p[command[2], command[3], command[4], command[5], command[6], command[7]])
      Case (caseValue=16)
        Script: movel_one_only(command[2],command[3])
      Case (caseValue=18)
        Script: movel_rot_only(command[2],command[3],command[4])
      Case (caseValue=20)
        Script: return_get_actual_joint_positions()
      Case (caseValue=21)
        Script: movej_ag([command[2], command[3], command[4], command[5], command[6], command[7]])
      Case (caseValue=22)
        Script: movel_ag(p[command[2], command[3], command[4], command[5], command[6], command[7]])
      Case (caseValue=25)
        Script: return_both_positions()
      Case (caseValue=30)
        Script: set_variable()
      Case (caseValue=35)
        Script: set_grind_variable()
      Case (caseValue=40)
        Script: grind()
      Case (caseValue=98)
        response := "socket reset"
      Case (caseValue=99)
        response := "exiting"
      Case (caseValue=2147483647)
        response := "unknown command"
    Script: command_finish()
    Set DigitalOutput pin=Stacklight; digitalValue=0
    If command[1]≟98
      Wait Sleep waitTime=0.5
      Script: socket_close()
      socket_is_open := False
    If command[1]≟99
      Wait Sleep waitTime=0.5
      Script: socket_close()
      socket_is_open := False
      Halt
  Else 
    Script: no_command()
